LIN {X 0,Y 382.998,Z 423.777,A -85,B 0,C 180,E1 -12171.424,E2 -12171.424} C_VEL
LIN {X 0,Y 383.055,Z 423.767,A -85,B 0,C 180,E1 -12174.96,E2 -12174.96} C_VEL
LIN {X 0,Y 383.051,Z 423.767,A -85,B 0,C 180,E1 -12175.302,E2 -12175.302} C_VEL
LIN {X 0,Y 382.387,Z 423.855,A -85,B 0,C 180,E1 -12176.18,E2 -12176.18} C_VEL
LIN {X 0,Y 379.5,Z 424.21,A -85,B 0,C 180,E1 -12177.606,E2 -12177.606} C_VEL
LIN {X 0,Y 377.061,Z 424.515,A -85,B 0,C 180,E1 -12178.76,E2 -12178.76} C_VEL
LIN {X 0,Y 376.028,Z 424.643,A -85,B 0,C 180,E1 -12179.652,E2 -12179.652} C_VEL
LIN {X 0,Y 375.952,Z 424.653,A -85,B 0,C 180,E1 -12179.955,E2 -12179.955} C_VEL
LIN {X 0,Y 375.955,Z 424.652,A -85,B 0,C 180,E1 -12182.828,E2 -12182.828} C_VEL
LIN {X 0,Y 375.962,Z 424.65,A -85,B 0,C 180,E1 -12185.415,E2 -12185.415} C_VEL
LIN {X 0,Y 375.978,Z 424.653,A -85,B 0,C 180,E1 -12188.27,E2 -12188.27} C_VEL
LIN {X 0,Y 375.938,Z 424.654,A -85,B 0,C 180,E1 -12191.601,E2 -12191.601} C_VEL
LIN {X 0,Y 375.932,Z 424.654,A -85,B 0,C 180,E1 -12195.268,E2 -12195.268} C_VEL
LIN {X 0,Y 375.938,Z 424.655,A -85,B 0,C 180,E1 -12198.399,E2 -12198.399} C_VEL
LIN {X 0,Y 375.978,Z 424.652,A -85,B 0,C 180,E1 -12201.73,E2 -12201.73} C_VEL
LIN {X 0,Y 375.984,Z 424.648,A -85,B 0,C 180,E1 -12205.333,E2 -12205.333} C_VEL
LIN {X 0,Y 375.962,Z 424.651,A -85,B 0,C 180,E1 -12208.438,E2 -12208.438} C_VEL
LIN {X 0,Y 376,Z 424.649,A -85,B 0,C 180,E1 -12212.141,E2 -12212.141} C_VEL
LIN {X 0,Y 376.009,Z 424.644,A -85,B 0,C 180,E1 -12214.539,E2 -12214.539} C_VEL
LIN {X 0,Y 375.962,Z 424.654,A -85,B 0,C 180,E1 -12218.045,E2 -12218.045} C_VEL
LIN {X 0,Y 376.028,Z 424.645,A -85,B 0,C 180,E1 -12221.474,E2 -12221.474} C_VEL
LIN {X 0,Y 376.074,Z 424.74,A -85,B 0,C 180,E1 -12224.034,E2 -12224.034} C_VEL
LIN {X 0,Y 378.978,Z 436.063,A -85,B 0,C 180,E1 -12224.952,E2 -12224.952} C_VEL
LIN {X 0,Y 379.745,Z 439.16,A -85,B 0,C 180,E1 -12225.24,E2 -12225.24} C_VEL
LIN {X 0,Y 379.247,Z 450.816,A -85,B 0,C 180,E1 -12226.333,E2 -12226.333} C_VEL
LIN {X 0,Y 378.652,Z 461.215,A -85,B 0,C 180,E1 -12227.539,E2 -12227.539} C_VEL
LIN {X 0,Y 377.962,Z 471.623,A -85,B 0,C 180,E1 -12229.012,E2 -12229.012} C_VEL
LIN {X 0,Y 377.299,Z 480.79,A -85,B 0,C 180,E1 -12230.627,E2 -12230.627} C_VEL
LIN {X 0,Y 376.92,Z 488.167,A -85,B 0,C 180,E1 -12232.231,E2 -12232.231} C_VEL
LIN {X 0,Y 376.501,Z 493.226,A -85,B 0,C 180,E1 -12233.569,E2 -12233.569} C_VEL
LIN {X 0,Y 376.262,Z 498.168,A -85,B 0,C 180,E1 -12235.178,E2 -12235.178} C_VEL
LIN {X 0,Y 375.83,Z 502.008,A -85,B 0,C 180,E1 -12236.784,E2 -12236.784} C_VEL
LIN {X 0,Y 375.952,Z 503.934,A -85,B 0,C 180,E1 -12237.857,E2 -12237.857} C_VEL
LIN {X 0,Y 375.864,Z 505.478,A -85,B 0,C 180,E1 -12238.928,E2 -12238.928} C_VEL
LIN {X 0,Y 375.983,Z 506.61,A -85,B 0,C 180,E1 -12240,E2 -12240} C_VEL
LIN {X 0,Y 376.041,Z 507.304,A -85,B 0,C 180,E1 -12241.071,E2 -12241.071} C_VEL
LIN {X 0,Y 376.261,Z 507.505,A -85,B 0,C 180,E1 -12243.212,E2 -12243.212} C_VEL
LIN {X 0,Y 376.364,Z 507.004,A -85,B 0,C 180,E1 -12244.283,E2 -12244.283} C_VEL
LIN {X 0,Y 376.837,Z 504.725,A -85,B 0,C 180,E1 -12246.425,E2 -12246.425} C_VEL
LIN {X 0,Y 377.509,Z 501.851,A -85,B 0,C 180,E1 -12248.026,E2 -12248.026} C_VEL
LIN {X 0,Y 378.12,Z 497.991,A -85,B 0,C 180,E1 -12249.63,E2 -12249.63} C_VEL
LIN {X 0,Y 378.925,Z 492.952,A -85,B 0,C 180,E1 -12251.23,E2 -12251.23} C_VEL
LIN {X 0,Y 379.835,Z 486.563,A -85,B 0,C 180,E1 -12252.828,E2 -12252.828} C_VEL
LIN {X 0,Y 380.937,Z 478.602,A -85,B 0,C 180,E1 -12254.422,E2 -12254.422} C_VEL
LIN {X 0,Y 381.922,Z 470.519,A -85,B 0,C 180,E1 -12255.749,E2 -12255.749} C_VEL
LIN {X 0,Y 383.075,Z 460.593,A -85,B 0,C 180,E1 -12257.07,E2 -12257.07} C_VEL
LIN {X 0,Y 384.276,Z 449.064,A -85,B 0,C 180,E1 -12258.3,E2 -12258.3} C_VEL
LIN {X 0,Y 384.418,Z 447.136,A -85,B 0,C 180,E1 -12258.479,E2 -12258.479} C_VEL
LIN {X 0,Y 380.901,Z 436.321,A -85,B 0,C 180,E1 -12259.779,E2 -12259.779} C_VEL
LIN {X 0,Y 376.958,Z 427.479,A -85,B 0,C 180,E1 -12260.81,E2 -12260.81} C_VEL
LIN {X 0,Y 375.977,Z 424.658,A -85,B 0,C 180,E1 -12261.095,E2 -12261.095} C_VEL
LIN {X 0,Y 375.997,Z 424.649,A -85,B 0,C 180,E1 -12264.281,E2 -12264.281} C_VEL
LIN {X 0,Y 376.023,Z 424.647,A -85,B 0,C 180,E1 -12266.652,E2 -12266.652} C_VEL
LIN {X 0,Y 375.973,Z 424.653,A -85,B 0,C 180,E1 -12269.079,E2 -12269.079} C_VEL
LIN {X 0,Y 375.952,Z 424.656,A -85,B 0,C 180,E1 -12272.828,E2 -12272.828} C_VEL
LIN {X 0,Y 375.96,Z 424.653,A -85,B 0,C 180,E1 -12275.415,E2 -12275.415} C_VEL
LIN {X 0,Y 375.976,Z 424.654,A -85,B 0,C 180,E1 -12278.27,E2 -12278.27} C_VEL
LIN {X 0,Y 375.937,Z 424.652,A -85,B 0,C 180,E1 -12281.601,E2 -12281.601} C_VEL
LIN {X 0,Y 375.997,Z 424.755,A -85,B 0,C 180,E1 -12284.798,E2 -12284.798} C_VEL
LIN {X 0,Y 377.748,Z 433.032,A -85,B 0,C 180,E1 -12288.09,E2 -12288.09} C_VEL
LIN {X 0,Y 379.603,Z 442.972,A -85,B 0,C 180,E1 -12291.746,E2 -12291.746} C_VEL
LIN {X 0,Y 379.908,Z 445.692,A -85,B 0,C 180,E1 -12292.7,E2 -12292.7} C_VEL
LIN {X 0,Y 378.943,Z 454.519,A -85,B 0,C 180,E1 -12295.551,E2 -12295.551} C_VEL
LIN {X 0,Y 377.958,Z 464.839,A -85,B 0,C 180,E1 -12298.799,E2 -12298.799} C_VEL
LIN {X 0,Y 377.121,Z 475.97,A -85,B 0,C 180,E1 -12302.231,E2 -12302.231} C_VEL
LIN {X 0,Y 376.225,Z 489.228,A -85,B 0,C 180,E1 -12306.254,E2 -12306.254} C_VEL
LIN {X 0,Y 375.618,Z 500.769,A -85,B 0,C 180,E1 -12309.75,E2 -12309.75} C_VEL
LIN {X 0,Y 377.668,Z 514.335,A -85,B 0,C 180,E1 -12310.571,E2 -12310.571} C_VEL
LIN {X 0,Y 379.007,Z 537.491,A -85,B 0,C 180,E1 -12312.078,E2 -12312.078} C_VEL
LIN {X 0,Y 379.272,Z 549.569,A -85,B 0,C 180,E1 -12313.031,E2 -12313.031} C_VEL
LIN {X 0,Y 378.26,Z 560.725,A -85,B 0,C 180,E1 -12314.094,E2 -12314.094} C_VEL
LIN {X 0,Y 377.222,Z 571.102,A -85,B 0,C 180,E1 -12315.336,E2 -12315.336} C_VEL
LIN {X 0,Y 376.519,Z 579.39,A -85,B 0,C 180,E1 -12316.542,E2 -12316.542} C_VEL
LIN {X 0,Y 375.778,Z 588.341,A -85,B 0,C 180,E1 -12318.128,E2 -12318.128} C_VEL
LIN {X 0,Y 375.246,Z 595.762,A -85,B 0,C 180,E1 -12319.751,E2 -12319.751} C_VEL
LIN {X 0,Y 375.084,Z 601.755,A -85,B 0,C 180,E1 -12321.379,E2 -12321.379} C_VEL
LIN {X 0,Y 375.1,Z 607.056,A -85,B 0,C 180,E1 -12323.23,E2 -12323.23} C_VEL
LIN {X 0,Y 375.181,Z 610.145,A -85,B 0,C 180,E1 -12324.625,E2 -12324.625} C_VEL
LIN {X 0,Y 375.348,Z 611.991,A -85,B 0,C 180,E1 -12325.705,E2 -12325.705} C_VEL
LIN {X 0,Y 375.389,Z 613.39,A -85,B 0,C 180,E1 -12326.78,E2 -12326.78} C_VEL
LIN {X 0,Y 375.732,Z 614.999,A -85,B 0,C 180,E1 -12328.928,E2 -12328.928} C_VEL
LIN {X 0,Y 375.771,Z 615.131,A -85,B 0,C 180,E1 -12330,E2 -12330} C_VEL
LIN {X 0,Y 375.738,Z 614.845,A -85,B 0,C 180,E1 -12331.072,E2 -12331.072} C_VEL
LIN {X 0,Y 375.423,Z 613.021,A -85,B 0,C 180,E1 -12333.219,E2 -12333.219} C_VEL
LIN {X 0,Y 375.326,Z 610.511,A -85,B 0,C 180,E1 -12334.833,E2 -12334.833} C_VEL
LIN {X 0,Y 375.17,Z 605.883,A -85,B 0,C 180,E1 -12336.859,E2 -12336.859} C_VEL
LIN {X 0,Y 375.149,Z 600.441,A -85,B 0,C 180,E1 -12338.619,E2 -12338.619} C_VEL
LIN {X 0,Y 375.319,Z 594.079,A -85,B 0,C 180,E1 -12340.247,E2 -12340.247} C_VEL
LIN {X 0,Y 375.769,Z 586.206,A -85,B 0,C 180,E1 -12341.872,E2 -12341.872} C_VEL
LIN {X 0,Y 376.443,Z 576.913,A -85,B 0,C 180,E1 -12343.41,E2 -12343.41} C_VEL
LIN {X 0,Y 376.946,Z 570.54,A -85,B 0,C 180,E1 -12344.302,E2 -12344.302} C_VEL
LIN {X 0,Y 377.832,Z 560.218,A -85,B 0,C 180,E1 -12345.509,E2 -12345.509} C_VEL
LIN {X 0,Y 378.693,Z 550.402,A -85,B 0,C 180,E1 -12346.44,E2 -12346.44} C_VEL
LIN {X 0,Y 378.312,Z 538.497,A -85,B 0,C 180,E1 -12347.378,E2 -12347.378} C_VEL
LIN {X 0,Y 377.647,Z 525.121,A -85,B 0,C 180,E1 -12348.193,E2 -12348.193} C_VEL
LIN {X 0,Y 376.458,Z 511.651,A -85,B 0,C 180,E1 -12348.786,E2 -12348.786} C_VEL
LIN {X 0,Y 375.446,Z 503.179,A -85,B 0,C 180,E1 -12349.087,E2 -12349.087} C_VEL
LIN {X 0,Y 375.935,Z 491.639,A -85,B 0,C 180,E1 -12352.534,E2 -12352.534} C_VEL
LIN {X 0,Y 376.689,Z 478.028,A -85,B 0,C 180,E1 -12356.601,E2 -12356.601} C_VEL
LIN {X 0,Y 377.67,Z 464.562,A -85,B 0,C 180,E1 -12360.662,E2 -12360.662} C_VEL
LIN {X 0,Y 378.648,Z 452.205,A -85,B 0,C 180,E1 -12364.479,E2 -12364.479} C_VEL
LIN {X 0,Y 379.451,Z 443.597,A -85,B 0,C 180,E1 -12367.21,E2 -12367.21} C_VEL
LIN {X 0,Y 378.303,Z 436.319,A -85,B 0,C 180,E1 -12369.732,E2 -12369.732} C_VEL
LIN {X 0,Y 376.689,Z 428.211,A -85,B 0,C 180,E1 -12372.709,E2 -12372.709} C_VEL
LIN {X 0,Y 375.986,Z 424.654,A -85,B 0,C 180,E1 -12374.131,E2 -12374.131} C_VEL
LIN {X 0,Y 375.932,Z 424.66,A -85,B 0,C 180,E1 -12377.7,E2 -12377.7} C_VEL
LIN {X 0,Y 375.965,Z 424.654,A -85,B 0,C 180,E1 -12380.538,E2 -12380.538} C_VEL
LIN {X 0,Y 375.965,Z 424.651,A -85,B 0,C 180,E1 -12383.495,E2 -12383.495} C_VEL
LIN {X 0,Y 375.963,Z 424.654,A -85,B 0,C 180,E1 -12385.889,E2 -12385.889} C_VEL
LIN {X 0,Y 375.965,Z 424.652,A -85,B 0,C 180,E1 -12389.687,E2 -12389.687} C_VEL
LIN {X 0,Y 376.02,Z 424.644,A -85,B 0,C 180,E1 -12393.348,E2 -12393.348} C_VEL
LIN {X 0,Y 375.997,Z 424.647,A -85,B 0,C 180,E1 -12396.888,E2 -12396.888} C_VEL
LIN {X 0,Y 375.999,Z 424.65,A -85,B 0,C 180,E1 -12400.339,E2 -12400.339} C_VEL
LIN {X 0,Y 376.03,Z 424.645,A -85,B 0,C 180,E1 -12403.719,E2 -12403.719} C_VEL
LIN {X 0,Y 376.108,Z 424.633,A -85,B 0,C 180,E1 -12407.042,E2 -12407.042} C_VEL
LIN {X 0,Y 376.119,Z 424.635,A -85,B 0,C 180,E1 -12410.319,E2 -12410.319} C_VEL
LIN {X 0,Y 376.234,Z 424.618,A -85,B 0,C 180,E1 -12413.565,E2 -12413.565} C_VEL
LIN {X 0,Y 376.356,Z 424.606,A -85,B 0,C 180,E1 -12417.86,E2 -12417.86} C_VEL
LIN {X 0,Y 376.491,Z 424.59,A -85,B 0,C 180,E1 -12420,E2 -12420} C_VEL
LIN {X 0,Y 376.186,Z 424.623,A -85,B 0,C 180,E1 -12423.213,E2 -12423.213} C_VEL
LIN {X 0,Y 376.235,Z 424.618,A -85,B 0,C 180,E1 -12426.639,E2 -12426.639} C_VEL
LIN {X 0,Y 376.207,Z 424.621,A -85,B 0,C 180,E1 -12428.595,E2 -12428.595} C_VEL
LIN {X 0,Y 376.052,Z 424.645,A -85,B 0,C 180,E1 -12431.864,E2 -12431.864} C_VEL
LIN {X 0,Y 376.06,Z 424.639,A -85,B 0,C 180,E1 -12435.168,E2 -12435.168} C_VEL
LIN {X 0,Y 376.025,Z 424.644,A -85,B 0,C 180,E1 -12438.526,E2 -12438.526} C_VEL
LIN {X 0,Y 375.965,Z 424.656,A -85,B 0,C 180,E1 -12441.954,E2 -12441.954} C_VEL
LIN {X 0,Y 376.008,Z 424.647,A -85,B 0,C 180,E1 -12445.461,E2 -12445.461} C_VEL
LIN {X 0,Y 375.962,Z 424.651,A -85,B 0,C 180,E1 -12449.08,E2 -12449.08} C_VEL
LIN {X 0,Y 375.952,Z 424.652,A -85,B 0,C 180,E1 -12452.829,E2 -12452.829} C_VEL
LIN {X 0,Y 375.96,Z 424.653,A -85,B 0,C 180,E1 -12455.416,E2 -12455.416} C_VEL
LIN {X 0,Y 375.978,Z 424.651,A -85,B 0,C 180,E1 -12458.271,E2 -12458.271} C_VEL
LIN {X 0,Y 375.937,Z 424.658,A -85,B 0,C 180,E1 -12461.601,E2 -12461.601} C_VEL
LIN {X 0,Y 375.932,Z 424.656,A -85,B 0,C 180,E1 -12465.268,E2 -12465.268} C_VEL
LIN {X 0,Y 375.937,Z 424.655,A -85,B 0,C 180,E1 -12468.399,E2 -12468.399} C_VEL
LIN {X 0,Y 375.978,Z 424.654,A -85,B 0,C 180,E1 -12471.729,E2 -12471.729} C_VEL
LIN {X 0,Y 375.983,Z 424.65,A -85,B 0,C 180,E1 -12475.333,E2 -12475.333} C_VEL
LIN {X 0,Y 375.979,Z 424.649,A -85,B 0,C 180,E1 -12478.44,E2 -12478.44} C_VEL
LIN {X 0,Y 376.005,Z 424.648,A -85,B 0,C 180,E1 -12482.142,E2 -12482.142} C_VEL
LIN {X 0,Y 376.009,Z 424.645,A -85,B 0,C 180,E1 -12484.539,E2 -12484.539} C_VEL
LIN {X 0,Y 375.967,Z 424.653,A -85,B 0,C 180,E1 -12488.046,E2 -12488.046} C_VEL
LIN {X 0,Y 376.028,Z 424.647,A -85,B 0,C 180,E1 -12491.474,E2 -12491.474} C_VEL
LIN {X 0,Y 376.066,Z 424.642,A -85,B 0,C 180,E1 -12494.961,E2 -12494.961} C_VEL
LIN {X 0,Y 379.867,Z 437.115,A -85,B 0,C 180,E1 -12495.996,E2 -12495.996} C_VEL
LIN {X 0,Y 381.449,Z 442.817,A -85,B 0,C 180,E1 -12496.549,E2 -12496.549} C_VEL
LIN {X 0,Y 380.847,Z 453.958,A -85,B 0,C 180,E1 -12497.613,E2 -12497.613} C_VEL
LIN {X 0,Y 380.009,Z 463.886,A -85,B 0,C 180,E1 -12498.783,E2 -12498.783} C_VEL
LIN {X 0,Y 379.149,Z 473.08,A -85,B 0,C 180,E1 -12500.127,E2 -12500.127} C_VEL
LIN {X 0,Y 378.39,Z 481.826,A -85,B 0,C 180,E1 -12501.724,E2 -12501.724} C_VEL
LIN {X 0,Y 377.633,Z 488.887,A -85,B 0,C 180,E1 -12503.321,E2 -12503.321} C_VEL
LIN {X 0,Y 377.166,Z 493.645,A -85,B 0,C 180,E1 -12504.654,E2 -12504.654} C_VEL
LIN {X 0,Y 376.746,Z 498.263,A -85,B 0,C 180,E1 -12506.257,E2 -12506.257} C_VEL
LIN {X 0,Y 376.324,Z 501.822,A -85,B 0,C 180,E1 -12507.86,E2 -12507.86} C_VEL
LIN {X 0,Y 376.142,Z 503.66,A -85,B 0,C 180,E1 -12508.93,E2 -12508.93} C_VEL
LIN {X 0,Y 376.055,Z 505.047,A -85,B 0,C 180,E1 -12510,E2 -12510} C_VEL
LIN {X 0,Y 375.934,Z 506.654,A -85,B 0,C 180,E1 -12512.143,E2 -12512.143} C_VEL
LIN {X 0,Y 375.812,Z 506.92,A -85,B 0,C 180,E1 -12513.216,E2 -12513.216} C_VEL
LIN {X 0,Y 375.896,Z 506.752,A -85,B 0,C 180,E1 -12514.289,E2 -12514.289} C_VEL
LIN {X 0,Y 376.335,Z 505.236,A -85,B 0,C 180,E1 -12516.434,E2 -12516.434} C_VEL
LIN {X 0,Y 376.464,Z 503.93,A -85,B 0,C 180,E1 -12517.509,E2 -12517.509} C_VEL
LIN {X 0,Y 376.828,Z 501.14,A -85,B 0,C 180,E1 -12519.122,E2 -12519.122} C_VEL
LIN {X 0,Y 377.389,Z 497.328,A -85,B 0,C 180,E1 -12520.733,E2 -12520.733} C_VEL
LIN {X 0,Y 377.993,Z 492.406,A -85,B 0,C 180,E1 -12522.347,E2 -12522.347} C_VEL
LIN {X 0,Y 378.625,Z 486.192,A -85,B 0,C 180,E1 -12523.964,E2 -12523.964} C_VEL
LIN {X 0,Y 379.358,Z 479.664,A -85,B 0,C 180,E1 -12525.34,E2 -12525.34} C_VEL
LIN {X 0,Y 380.387,Z 470.371,A -85,B 0,C 180,E1 -12526.918,E2 -12526.918} C_VEL
LIN {X 0,Y 381.256,Z 460.584,A -85,B 0,C 180,E1 -12528.263,E2 -12528.263} C_VEL
LIN {X 0,Y 382.202,Z 449.737,A -85,B 0,C 180,E1 -12529.441,E2 -12529.441} C_VEL
LIN {X 0,Y 382.437,Z 444.949,A -85,B 0,C 180,E1 -12529.889,E2 -12529.889} C_VEL
LIN {X 0,Y 379.598,Z 435.417,A -85,B 0,C 180,E1 -12530.857,E2 -12530.857} C_VEL
LIN {X 0,Y 375.965,Z 424.653,A -85,B 0,C 180,E1 -12531.8,E2 -12531.8} C_VEL
LIN {X 0,Y 376.01,Z 424.644,A -85,B 0,C 180,E1 -12535.461,E2 -12535.461} C_VEL
LIN {X 0,Y 375.975,Z 424.648,A -85,B 0,C 180,E1 -12539.079,E2 -12539.079} C_VEL
LIN {X 0,Y 375.952,Z 424.653,A -85,B 0,C 180,E1 -12539.955,E2 -12539.955} C_VEL
LIN {X 0,Y 375.295,Z 424.74,A -85,B 0,C 180,E1 -12540.849,E2 -12540.849} C_VEL
LIN {X 0,Y 372.41,Z 425.098,A -85,B 0,C 180,E1 -12542.304,E2 -12542.304} C_VEL
LIN {X 0,Y 369.985,Z 425.395,A -85,B 0,C 180,E1 -12543.48,E2 -12543.48} C_VEL
LIN {X 0,Y 368.985,Z 425.523,A -85,B 0,C 180,E1 -12544.39,E2 -12544.39} C_VEL
LIN {X 0,Y 368.926,Z 425.526,A -85,B 0,C 180,E1 -12544.698,E2 -12544.698} C_VEL
LIN {X 0,Y 368.908,Z 425.53,A -85,B 0,C 180,E1 -12547.563,E2 -12547.563} C_VEL
LIN {X 0,Y 368.915,Z 425.532,A -85,B 0,C 180,E1 -12550.37,E2 -12550.37} C_VEL
LIN {X 0,Y 368.887,Z 425.533,A -85,B 0,C 180,E1 -12553.616,E2 -12553.616} C_VEL
LIN {X 0,Y 368.89,Z 425.532,A -85,B 0,C 180,E1 -12556.696,E2 -12556.696} C_VEL
LIN {X 0,Y 368.915,Z 425.53,A -85,B 0,C 180,E1 -12559.643,E2 -12559.643} C_VEL
LIN {X 0,Y 368.905,Z 425.529,A -85,B 0,C 180,E1 -12563.144,E2 -12563.144} C_VEL
LIN {X 0,Y 368.902,Z 425.531,A -85,B 0,C 180,E1 -12566.462,E2 -12566.462} C_VEL
LIN {X 0,Y 368.933,Z 425.526,A -85,B 0,C 180,E1 -12569.046,E2 -12569.046} C_VEL
LIN {X 0,Y 368.984,Z 425.522,A -85,B 0,C 180,E1 -12571.564,E2 -12571.564} C_VEL
LIN {X 0,Y 369.004,Z 425.521,A -85,B 0,C 180,E1 -12574.02,E2 -12574.02} C_VEL
LIN {X 0,Y 368.929,Z 425.53,A -85,B 0,C 180,E1 -12577.604,E2 -12577.604} C_VEL
LIN {X 0,Y 368.986,Z 425.52,A -85,B 0,C 180,E1 -12581.107,E2 -12581.107} C_VEL
LIN {X 0,Y 369.03,Z 425.519,A -85,B 0,C 180,E1 -12583.792,E2 -12583.792} C_VEL
LIN {X 0,Y 372.433,Z 438.96,A -85,B 0,C 180,E1 -12584.943,E2 -12584.943} C_VEL
LIN {X 0,Y 372.839,Z 441.474,A -85,B 0,C 180,E1 -12585.174,E2 -12585.174} C_VEL
LIN {X 0,Y 372.139,Z 453.389,A -85,B 0,C 180,E1 -12586.345,E2 -12586.345} C_VEL
LIN {X 0,Y 371.612,Z 463.54,A -85,B 0,C 180,E1 -12587.577,E2 -12587.577} C_VEL
LIN {X 0,Y 370.995,Z 471.979,A -85,B 0,C 180,E1 -12588.803,E2 -12588.803} C_VEL
LIN {X 0,Y 370.312,Z 481.384,A -85,B 0,C 180,E1 -12590.472,E2 -12590.472} C_VEL
LIN {X 0,Y 369.919,Z 488.736,A -85,B 0,C 180,E1 -12592.083,E2 -12592.083} C_VEL
LIN {X 0,Y 369.482,Z 493.875,A -85,B 0,C 180,E1 -12593.446,E2 -12593.446} C_VEL
LIN {X 0,Y 369.232,Z 498.907,A -85,B 0,C 180,E1 -12595.086,E2 -12595.086} C_VEL
LIN {X 0,Y 368.792,Z 502.844,A -85,B 0,C 180,E1 -12596.722,E2 -12596.722} C_VEL
LIN {X 0,Y 368.927,Z 504.844,A -85,B 0,C 180,E1 -12597.816,E2 -12597.816} C_VEL
LIN {X 0,Y 368.84,Z 506.432,A -85,B 0,C 180,E1 -12598.908,E2 -12598.908} C_VEL
LIN {X 0,Y 368.966,Z 507.61,A -85,B 0,C 180,E1 -12600,E2 -12600} C_VEL
LIN {X 0,Y 369.028,Z 508.374,A -85,B 0,C 180,E1 -12601.091,E2 -12601.091} C_VEL
LIN {X 0,Y 369.152,Z 508.703,A -85,B 0,C 180,E1 -12602.182,E2 -12602.182} C_VEL
LIN {X 0,Y 369.275,Z 508.653,A -85,B 0,C 180,E1 -12603.273,E2 -12603.273} C_VEL
LIN {X 0,Y 369.385,Z 508.216,A -85,B 0,C 180,E1 -12604.365,E2 -12604.365} C_VEL
LIN {X 0,Y 369.905,Z 506.039,A -85,B 0,C 180,E1 -12606.546,E2 -12606.546} C_VEL
LIN {X 0,Y 370.63,Z 503.262,A -85,B 0,C 180,E1 -12608.176,E2 -12608.176} C_VEL
LIN {X 0,Y 371.28,Z 499.481,A -85,B 0,C 180,E1 -12609.809,E2 -12609.809} C_VEL
LIN {X 0,Y 372.146,Z 494.534,A -85,B 0,C 180,E1 -12611.437,E2 -12611.437} C_VEL
LIN {X 0,Y 373.133,Z 488.278,A -85,B 0,C 180,E1 -12613.063,E2 -12613.063} C_VEL
LIN {X 0,Y 374.328,Z 480.505,A -85,B 0,C 180,E1 -12614.682,E2 -12614.682} C_VEL
LIN {X 0,Y 375.379,Z 472.598,A -85,B 0,C 180,E1 -12616.031,E2 -12616.031} C_VEL
LIN {X 0,Y 376.589,Z 462.892,A -85,B 0,C 180,E1 -12617.373,E2 -12617.373} C_VEL
LIN {X 0,Y 377.874,Z 451.542,A -85,B 0,C 180,E1 -12618.641,E2 -12618.641} C_VEL
LIN {X 0,Y 378.064,Z 449.476,A -85,B 0,C 180,E1 -12618.84,E2 -12618.84} C_VEL
LIN {X 0,Y 375.264,Z 440.491,A -85,B 0,C 180,E1 -12619.986,E2 -12619.986} C_VEL
LIN {X 0,Y 370.695,Z 429.697,A -85,B 0,C 180,E1 -12621.328,E2 -12621.328} C_VEL
LIN {X 0,Y 369.043,Z 426.27,A -85,B 0,C 180,E1 -12621.741,E2 -12621.741} C_VEL
LIN {X 0,Y 368.941,Z 425.536,A -85,B 0,C 180,E1 -12621.805,E2 -12621.805} C_VEL
LIN {X 0,Y 368.961,Z 425.527,A -85,B 0,C 180,E1 -12624.775,E2 -12624.775} C_VEL
LIN {X 0,Y 368.971,Z 425.526,A -85,B 0,C 180,E1 -12627.203,E2 -12627.203} C_VEL
LIN {X 0,Y 368.922,Z 425.529,A -85,B 0,C 180,E1 -12629.69,E2 -12629.69} C_VEL
LIN {X 0,Y 368.9,Z 425.533,A -85,B 0,C 180,E1 -12633.043,E2 -12633.043} C_VEL
LIN {X 0,Y 368.92,Z 425.532,A -85,B 0,C 180,E1 -12636.197,E2 -12636.197} C_VEL
LIN {X 0,Y 368.905,Z 425.532,A -85,B 0,C 180,E1 -12638.953,E2 -12638.953} C_VEL
LIN {X 0,Y 368.883,Z 425.531,A -85,B 0,C 180,E1 -12642.009,E2 -12642.009} C_VEL
LIN {X 0,Y 368.924,Z 425.588,A -85,B 0,C 180,E1 -12644.328,E2 -12644.328} C_VEL
LIN {X 0,Y 370.894,Z 434.784,A -85,B 0,C 180,E1 -12648.077,E2 -12648.077} C_VEL
LIN {X 0,Y 372.544,Z 443.871,A -85,B 0,C 180,E1 -12651.498,E2 -12651.498} C_VEL
LIN {X 0,Y 372.941,Z 446.174,A -85,B 0,C 180,E1 -12652.324,E2 -12652.324} C_VEL
LIN {X 0,Y 372.168,Z 453.768,A -85,B 0,C 180,E1 -12654.853,E2 -12654.853} C_VEL
LIN {X 0,Y 371.047,Z 464.964,A -85,B 0,C 180,E1 -12658.468,E2 -12658.468} C_VEL
LIN {X 0,Y 370.034,Z 477.018,A -85,B 0,C 180,E1 -12662.268,E2 -12662.268} C_VEL
LIN {X 0,Y 369.173,Z 489.138,A -85,B 0,C 180,E1 -12666.034,E2 -12666.034} C_VEL
LIN {X 0,Y 368.627,Z 499.227,A -85,B 0,C 180,E1 -12669.1,E2 -12669.1} C_VEL
LIN {X 0,Y 370.992,Z 513.976,A -85,B 0,C 180,E1 -12670.063,E2 -12670.063} C_VEL
LIN {X 0,Y 371.818,Z 528.383,A -85,B 0,C 180,E1 -12671.106,E2 -12671.106} C_VEL
LIN {X 0,Y 372.226,Z 545.56,A -85,B 0,C 180,E1 -12672.416,E2 -12672.416} C_VEL
LIN {X 0,Y 372.14,Z 553.252,A -85,B 0,C 180,E1 -12673.12,E2 -12673.12} C_VEL
LIN {X 0,Y 370.857,Z 564.617,A -85,B 0,C 180,E1 -12674.333,E2 -12674.333} C_VEL
LIN {X 0,Y 369.827,Z 575.003,A -85,B 0,C 180,E1 -12675.738,E2 -12675.738} C_VEL
LIN {X 0,Y 369.136,Z 583.091,A -85,B 0,C 180,E1 -12677.073,E2 -12677.073} C_VEL
LIN {X 0,Y 368.46,Z 591.318,A -85,B 0,C 180,E1 -12678.725,E2 -12678.725} C_VEL
LIN {X 0,Y 368.123,Z 596.936,A -85,B 0,C 180,E1 -12680.106,E2 -12680.106} C_VEL
LIN {X 0,Y 368.006,Z 602.482,A -85,B 0,C 180,E1 -12681.765,E2 -12681.765} C_VEL
LIN {X 0,Y 368.058,Z 606.842,A -85,B 0,C 180,E1 -12683.421,E2 -12683.421} C_VEL
LIN {X 0,Y 368.111,Z 609.161,A -85,B 0,C 180,E1 -12684.522,E2 -12684.522} C_VEL
LIN {X 0,Y 368.277,Z 610.998,A -85,B 0,C 180,E1 -12685.622,E2 -12685.622} C_VEL
LIN {X 0,Y 368.339,Z 612.395,A -85,B 0,C 180,E1 -12686.718,E2 -12686.718} C_VEL
LIN {X 0,Y 368.702,Z 613.992,A -85,B 0,C 180,E1 -12688.908,E2 -12688.908} C_VEL
LIN {X 0,Y 368.748,Z 614.116,A -85,B 0,C 180,E1 -12690,E2 -12690} C_VEL
LIN {X 0,Y 368.709,Z 613.822,A -85,B 0,C 180,E1 -12691.092,E2 -12691.092} C_VEL
LIN {X 0,Y 368.38,Z 611.98,A -85,B 0,C 180,E1 -12693.281,E2 -12693.281} C_VEL
LIN {X 0,Y 368.266,Z 609.455,A -85,B 0,C 180,E1 -12694.926,E2 -12694.926} C_VEL
LIN {X 0,Y 368.097,Z 605.135,A -85,B 0,C 180,E1 -12696.866,E2 -12696.866} C_VEL
LIN {X 0,Y 368.072,Z 599.336,A -85,B 0,C 180,E1 -12698.786,E2 -12698.786} C_VEL
LIN {X 0,Y 368.258,Z 592.954,A -85,B 0,C 180,E1 -12700.445,E2 -12700.445} C_VEL
LIN {X 0,Y 368.76,Z 585.055,A -85,B 0,C 180,E1 -12702.101,E2 -12702.101} C_VEL
LIN {X 0,Y 369.373,Z 576.241,A -85,B 0,C 180,E1 -12703.592,E2 -12703.592} C_VEL
LIN {X 0,Y 370.252,Z 567.196,A -85,B 0,C 180,E1 -12704.848,E2 -12704.848} C_VEL
LIN {X 0,Y 371.163,Z 556.345,A -85,B 0,C 180,E1 -12706.077,E2 -12706.077} C_VEL
LIN {X 0,Y 371.695,Z 549.079,A -85,B 0,C 180,E1 -12706.759,E2 -12706.759} C_VEL
LIN {X 0,Y 371.319,Z 537.235,A -85,B 0,C 180,E1 -12707.707,E2 -12707.707} C_VEL
LIN {X 0,Y 370.607,Z 524.052,A -85,B 0,C 180,E1 -12708.527,E2 -12708.527} C_VEL
LIN {X 0,Y 369.414,Z 510.776,A -85,B 0,C 180,E1 -12709.126,E2 -12709.126} C_VEL
LIN {X 0,Y 368.408,Z 502.192,A -85,B 0,C 180,E1 -12709.429,E2 -12709.429} C_VEL
LIN {X 0,Y 368.901,Z 490.544,A -85,B 0,C 180,E1 -12712.989,E2 -12712.989} C_VEL
LIN {X 0,Y 369.64,Z 478.527,A -85,B 0,C 180,E1 -12716.669,E2 -12716.669} C_VEL
LIN {X 0,Y 370.643,Z 465.167,A -85,B 0,C 180,E1 -12720.795,E2 -12720.795} C_VEL
LIN {X 0,Y 371.651,Z 453.24,A -85,B 0,C 180,E1 -12724.562,E2 -12724.562} C_VEL
LIN {X 0,Y 372.461,Z 445.265,A -85,B 0,C 180,E1 -12727.143,E2 -12727.143} C_VEL
LIN {X 0,Y 371.689,Z 439.455,A -85,B 0,C 180,E1 -12729.173,E2 -12729.173} C_VEL
LIN {X 0,Y 370.092,Z 431.225,A -85,B 0,C 180,E1 -12732.217,E2 -12732.217} C_VEL
LIN {X 0,Y 368.917,Z 425.537,A -85,B 0,C 180,E1 -12734.501,E2 -12734.501} C_VEL
LIN {X 0,Y 368.884,Z 425.538,A -85,B 0,C 180,E1 -12738.178,E2 -12738.178} C_VEL
LIN {X 0,Y 368.911,Z 425.529,A -85,B 0,C 180,E1 -12741.359,E2 -12741.359} C_VEL
LIN {X 0,Y 368.937,Z 425.525,A -85,B 0,C 180,E1 -12745.147,E2 -12745.147} C_VEL
LIN {X 0,Y 368.929,Z 425.527,A -85,B 0,C 180,E1 -12749.047,E2 -12749.047} C_VEL
LIN {X 0,Y 368.964,Z 425.523,A -85,B 0,C 180,E1 -12752.797,E2 -12752.797} C_VEL
LIN {X 0,Y 368.946,Z 425.53,A -85,B 0,C 180,E1 -12756.113,E2 -12756.113} C_VEL
LIN {X 0,Y 368.938,Z 425.53,A -85,B 0,C 180,E1 -12759.947,E2 -12759.947} C_VEL
LIN {X 0,Y 368.977,Z 425.521,A -85,B 0,C 180,E1 -12763.399,E2 -12763.399} C_VEL
LIN {X 0,Y 369.061,Z 425.511,A -85,B 0,C 180,E1 -12766.79,E2 -12766.79} C_VEL
LIN {X 0,Y 369.069,Z 425.515,A -85,B 0,C 180,E1 -12770.132,E2 -12770.132} C_VEL
LIN {X 0,Y 369.192,Z 425.494,A -85,B 0,C 180,E1 -12773.442,E2 -12773.442} C_VEL
LIN {X 0,Y 369.321,Z 425.482,A -85,B 0,C 180,E1 -12777.819,E2 -12777.819} C_VEL
LIN {X 0,Y 369.46,Z 425.466,A -85,B 0,C 180,E1 -12780,E2 -12780} C_VEL
LIN {X 0,Y 369.318,Z 425.483,A -85,B 0,C 180,E1 -12782.181,E2 -12782.181} C_VEL
LIN {X 0,Y 369.205,Z 425.493,A -85,B 0,C 180,E1 -12786.627,E2 -12786.627} C_VEL
LIN {X 0,Y 369.139,Z 425.501,A -85,B 0,C 180,E1 -12788.761,E2 -12788.761} C_VEL
LIN {X 0,Y 369.008,Z 425.522,A -85,B 0,C 180,E1 -12792.093,E2 -12792.093} C_VEL
LIN {X 0,Y 368.999,Z 425.519,A -85,B 0,C 180,E1 -12795.465,E2 -12795.465} C_VEL
LIN {X 0,Y 368.984,Z 425.52,A -85,B 0,C 180,E1 -12798.893,E2 -12798.893} C_VEL
LIN {X 0,Y 368.934,Z 425.528,A -85,B 0,C 180,E1 -12802.395,E2 -12802.395} C_VEL
LIN {X 0,Y 369.001,Z 425.523,A -85,B 0,C 180,E1 -12805.98,E2 -12805.98} C_VEL
LIN {X 0,Y 368.916,Z 425.532,A -85,B 0,C 180,E1 -12809.691,E2 -12809.691} C_VEL
LIN {X 0,Y 368.9,Z 425.53,A -85,B 0,C 180,E1 -12813.044,E2 -12813.044} C_VEL
LIN {X 0,Y 368.92,Z 425.531,A -85,B 0,C 180,E1 -12816.197,E2 -12816.197} C_VEL
LIN {X 0,Y 368.906,Z 425.529,A -85,B 0,C 180,E1 -12818.953,E2 -12818.953} C_VEL
LIN {X 0,Y 368.884,Z 425.537,A -85,B 0,C 180,E1 -12822.01,E2 -12822.01} C_VEL
LIN {X 0,Y 368.885,Z 425.533,A -85,B 0,C 180,E1 -12825.177,E2 -12825.177} C_VEL
LIN {X 0,Y 368.886,Z 425.535,A -85,B 0,C 180,E1 -12828.178,E2 -12828.178} C_VEL
LIN {X 0,Y 368.912,Z 425.531,A -85,B 0,C 180,E1 -12831.36,E2 -12831.36} C_VEL
LIN {X 0,Y 368.939,Z 425.526,A -85,B 0,C 180,E1 -12835.147,E2 -12835.147} C_VEL
LIN {X 0,Y 368.932,Z 425.527,A -85,B 0,C 180,E1 -12839.047,E2 -12839.047} C_VEL
LIN {X 0,Y 368.99,Z 425.524,A -85,B 0,C 180,E1 -12841.565,E2 -12841.565} C_VEL
LIN {X 0,Y 368.961,Z 425.524,A -85,B 0,C 180,E1 -12845.225,E2 -12845.225} C_VEL
LIN {X 0,Y 368.941,Z 425.526,A -85,B 0,C 180,E1 -12848.974,E2 -12848.974} C_VEL
LIN {X 0,Y 368.994,Z 425.52,A -85,B 0,C 180,E1 -12852.258,E2 -12852.258} C_VEL
LIN {X 0,Y 369.027,Z 425.634,A -85,B 0,C 180,E1 -12854.635,E2 -12854.635} C_VEL
LIN {X 0,Y 372.753,Z 437.637,A -85,B 0,C 180,E1 -12855.642,E2 -12855.642} C_VEL
LIN {X 0,Y 374.612,Z 444.234,A -85,B 0,C 180,E1 -12856.299,E2 -12856.299} C_VEL
LIN {X 0,Y 374.014,Z 455.295,A -85,B 0,C 180,E1 -12857.383,E2 -12857.383} C_VEL
LIN {X 0,Y 373.149,Z 465.158,A -85,B 0,C 180,E1 -12858.574,E2 -12858.574} C_VEL
LIN {X 0,Y 372.253,Z 474.295,A -85,B 0,C 180,E1 -12859.943,E2 -12859.943} C_VEL
LIN {X 0,Y 371.461,Z 483.007,A -85,B 0,C 180,E1 -12861.569,E2 -12861.569} C_VEL
LIN {X 0,Y 370.672,Z 490.038,A -85,B 0,C 180,E1 -12863.195,E2 -12863.195} C_VEL
LIN {X 0,Y 370.213,Z 494.765,A -85,B 0,C 180,E1 -12864.554,E2 -12864.554} C_VEL
LIN {X 0,Y 369.753,Z 499.363,A -85,B 0,C 180,E1 -12866.186,E2 -12866.186} C_VEL
LIN {X 0,Y 369.308,Z 502.901,A -85,B 0,C 180,E1 -12867.819,E2 -12867.819} C_VEL
LIN {X 0,Y 369.121,Z 504.726,A -85,B 0,C 180,E1 -12868.909,E2 -12868.909} C_VEL
LIN {X 0,Y 368.981,Z 507.069,A -85,B 0,C 180,E1 -12871.092,E2 -12871.092} C_VEL
LIN {X 0,Y 368.91,Z 507.681,A -85,B 0,C 180,E1 -12872.184,E2 -12872.184} C_VEL
LIN {X 0,Y 368.788,Z 507.936,A -85,B 0,C 180,E1 -12873.278,E2 -12873.278} C_VEL
LIN {X 0,Y 369.046,Z 507.174,A -85,B 0,C 180,E1 -12875.464,E2 -12875.464} C_VEL
LIN {X 0,Y 369.346,Z 506.212,A -85,B 0,C 180,E1 -12876.556,E2 -12876.556} C_VEL
LIN {X 0,Y 369.488,Z 504.894,A -85,B 0,C 180,E1 -12877.652,E2 -12877.652} C_VEL
LIN {X 0,Y 369.885,Z 502.085,A -85,B 0,C 180,E1 -12879.294,E2 -12879.294} C_VEL
LIN {X 0,Y 370.461,Z 498.252,A -85,B 0,C 180,E1 -12880.936,E2 -12880.936} C_VEL
LIN {X 0,Y 371.11,Z 493.303,A -85,B 0,C 180,E1 -12882.579,E2 -12882.579} C_VEL
LIN {X 0,Y 371.786,Z 487.049,A -85,B 0,C 180,E1 -12884.226,E2 -12884.226} C_VEL
LIN {X 0,Y 372.777,Z 478.774,A -85,B 0,C 180,E1 -12885.947,E2 -12885.947} C_VEL
LIN {X 0,Y 373.83,Z 469.381,A -85,B 0,C 180,E1 -12887.506,E2 -12887.506} C_VEL
LIN {X 0,Y 374.67,Z 460.177,A -85,B 0,C 180,E1 -12888.738,E2 -12888.738} C_VEL
LIN {X 0,Y 375.601,Z 449.67,A -85,B 0,C 180,E1 -12889.869,E2 -12889.869} C_VEL
LIN {X 0,Y 375.713,Z 446.52,A -85,B 0,C 180,E1 -12890.174,E2 -12890.174} C_VEL
LIN {X 0,Y 372.201,Z 435.095,A -85,B 0,C 180,E1 -12891.357,E2 -12891.357} C_VEL
LIN {X 0,Y 368.924,Z 425.532,A -85,B 0,C 180,E1 -12892.215,E2 -12892.215} C_VEL
LIN {X 0,Y 369.004,Z 425.52,A -85,B 0,C 180,E1 -12895.98,E2 -12895.98} C_VEL
LIN {X 0,Y 368.965,Z 425.523,A -85,B 0,C 180,E1 -12898.812,E2 -12898.812} C_VEL
LIN {X 0,Y 368.903,Z 425.536,A -85,B 0,C 180,E1 -12902.238,E2 -12902.238} C_VEL
LIN {X 0,Y 368.926,Z 425.526,A -85,B 0,C 180,E1 -12904.698,E2 -12904.698} C_VEL
LIN {X 0,Y 368.314,Z 425.606,A -85,B 0,C 180,E1 -12905.609,E2 -12905.609} C_VEL
LIN {X 0,Y 365.457,Z 425.961,A -85,B 0,C 180,E1 -12907.089,E2 -12907.089} C_VEL
LIN {X 0,Y 362.999,Z 426.27,A -85,B 0,C 180,E1 -12908.286,E2 -12908.286} C_VEL
LIN {X 0,Y 361.941,Z 426.397,A -85,B 0,C 180,E1 -12909.213,E2 -12909.213} C_VEL
LIN {X 0,Y 361.855,Z 426.408,A -85,B 0,C 180,E1 -12909.527,E2 -12909.527} C_VEL
LIN {X 0,Y 361.84,Z 426.409,A -85,B 0,C 180,E1 -12912.829,E2 -12912.829} C_VEL
LIN {X 0,Y 361.823,Z 426.416,A -85,B 0,C 180,E1 -12915.946,E2 -12915.946} C_VEL
LIN {X 0,Y 361.839,Z 426.409,A -85,B 0,C 180,E1 -12919.245,E2 -12919.245} C_VEL
LIN {X 0,Y 361.868,Z 426.406,A -85,B 0,C 180,E1 -12922.777,E2 -12922.777} C_VEL
LIN {X 0,Y 361.859,Z 426.411,A -85,B 0,C 180,E1 -12925.72,E2 -12925.72} C_VEL
LIN {X 0,Y 361.879,Z 426.408,A -85,B 0,C 180,E1 -12929.672,E2 -12929.672} C_VEL
LIN {X 0,Y 361.958,Z 426.397,A -85,B 0,C 180,E1 -12933.475,E2 -12933.475} C_VEL
LIN {X 0,Y 361.886,Z 426.404,A -85,B 0,C 180,E1 -12937.144,E2 -12937.144} C_VEL
LIN {X 0,Y 361.925,Z 426.398,A -85,B 0,C 180,E1 -12940.724,E2 -12940.724} C_VEL
LIN {X 0,Y 361.995,Z 426.431,A -85,B 0,C 180,E1 -12943.613,E2 -12943.613} C_VEL
LIN {X 0,Y 365.046,Z 438.518,A -85,B 0,C 180,E1 -12944.631,E2 -12944.631} C_VEL
LIN {X 0,Y 365.865,Z 442.716,A -85,B 0,C 180,E1 -12945.029,E2 -12945.029} C_VEL
LIN {X 0,Y 365.138,Z 454.527,A -85,B 0,C 180,E1 -12946.22,E2 -12946.22} C_VEL
LIN {X 0,Y 364.597,Z 464.649,A -85,B 0,C 180,E1 -12947.475,E2 -12947.475} C_VEL
LIN {X 0,Y 363.895,Z 473.92,A -85,B 0,C 180,E1 -12948.864,E2 -12948.864} C_VEL
LIN {X 0,Y 363.316,Z 481.97,A -85,B 0,C 180,E1 -12950.324,E2 -12950.324} C_VEL
LIN {X 0,Y 362.919,Z 489.262,A -85,B 0,C 180,E1 -12951.929,E2 -12951.929} C_VEL
LIN {X 0,Y 362.466,Z 494.509,A -85,B 0,C 180,E1 -12953.319,E2 -12953.319} C_VEL
LIN {X 0,Y 362.208,Z 499.641,A -85,B 0,C 180,E1 -12954.991,E2 -12954.991} C_VEL
LIN {X 0,Y 361.753,Z 503.673,A -85,B 0,C 180,E1 -12956.659,E2 -12956.659} C_VEL
LIN {X 0,Y 361.9,Z 505.752,A -85,B 0,C 180,E1 -12957.774,E2 -12957.774} C_VEL
LIN {X 0,Y 361.815,Z 507.389,A -85,B 0,C 180,E1 -12958.887,E2 -12958.887} C_VEL
LIN {X 0,Y 361.948,Z 508.605,A -85,B 0,C 180,E1 -12960,E2 -12960} C_VEL
LIN {X 0,Y 362.014,Z 509.44,A -85,B 0,C 180,E1 -12961.112,E2 -12961.112} C_VEL
LIN {X 0,Y 362.146,Z 509.822,A -85,B 0,C 180,E1 -12962.224,E2 -12962.224} C_VEL
LIN {X 0,Y 362.434,Z 509.442,A -85,B 0,C 180,E1 -12964.448,E2 -12964.448} C_VEL
LIN {X 0,Y 362.674,Z 508.617,A -85,B 0,C 180,E1 -12965.56,E2 -12965.56} C_VEL
LIN {X 0,Y 362.992,Z 507.372,A -85,B 0,C 180,E1 -12966.671,E2 -12966.671} C_VEL
LIN {X 0,Y 363.748,Z 504.674,A -85,B 0,C 180,E1 -12968.332,E2 -12968.332} C_VEL
LIN {X 0,Y 364.446,Z 500.985,A -85,B 0,C 180,E1 -12969.995,E2 -12969.995} C_VEL
LIN {X 0,Y 365.393,Z 496.173,A -85,B 0,C 180,E1 -12971.651,E2 -12971.651} C_VEL
LIN {X 0,Y 366.467,Z 490.095,A -85,B 0,C 180,E1 -12973.305,E2 -12973.305} C_VEL
LIN {X 0,Y 367.728,Z 482.439,A -85,B 0,C 180,E1 -12974.952,E2 -12974.952} C_VEL
LIN {X 0,Y 369.078,Z 472.99,A -85,B 0,C 180,E1 -12976.596,E2 -12976.596} C_VEL
LIN {X 0,Y 370.322,Z 463.898,A -85,B 0,C 180,E1 -12977.87,E2 -12977.87} C_VEL
LIN {X 0,Y 371.745,Z 452.318,A -85,B 0,C 180,E1 -12979.179,E2 -12979.179} C_VEL
LIN {X 0,Y 369.318,Z 443.699,A -85,B 0,C 180,E1 -12980.322,E2 -12980.322} C_VEL
LIN {X 0,Y 365.526,Z 434.468,A -85,B 0,C 180,E1 -12981.55,E2 -12981.55} C_VEL
LIN {X 0,Y 362.211,Z 427.729,A -85,B 0,C 180,E1 -12982.449,E2 -12982.449} C_VEL
LIN {X 0,Y 361.9,Z 426.408,A -85,B 0,C 180,E1 -12982.591,E2 -12982.591} C_VEL
LIN {X 0,Y 361.958,Z 426.398,A -85,B 0,C 180,E1 -12986.525,E2 -12986.525} C_VEL
LIN {X 0,Y 361.877,Z 426.409,A -85,B 0,C 180,E1 -12990.328,E2 -12990.328} C_VEL
LIN {X 0,Y 361.857,Z 426.412,A -85,B 0,C 180,E1 -12994.28,E2 -12994.28} C_VEL
LIN {X 0,Y 361.866,Z 426.408,A -85,B 0,C 180,E1 -12997.223,E2 -12997.223} C_VEL
LIN {X 0,Y 361.838,Z 426.413,A -85,B 0,C 180,E1 -13000.755,E2 -13000.755} C_VEL
LIN {X 0,Y 361.86,Z 426.437,A -85,B 0,C 180,E1 -13003.868,E2 -13003.868} C_VEL
LIN {X 0,Y 363.672,Z 434.964,A -85,B 0,C 180,E1 -13007.438,E2 -13007.438} C_VEL
LIN {X 0,Y 365.396,Z 444.028,A -85,B 0,C 180,E1 -13010.956,E2 -13010.956} C_VEL
LIN {X 0,Y 365.907,Z 447.054,A -85,B 0,C 180,E1 -13012.075,E2 -13012.075} C_VEL
LIN {X 0,Y 365.706,Z 450.95,A -85,B 0,C 180,E1 -13013.434,E2 -13013.434} C_VEL
LIN {X 0,Y 364.396,Z 462.6,A -85,B 0,C 180,E1 -13017.314,E2 -13017.314} C_VEL
LIN {X 0,Y 363.27,Z 474.195,A -85,B 0,C 180,E1 -13021.075,E2 -13021.075} C_VEL
LIN {X 0,Y 362.371,Z 485.688,A -85,B 0,C 180,E1 -13024.743,E2 -13024.743} C_VEL
LIN {X 0,Y 361.644,Z 497.073,A -85,B 0,C 180,E1 -13028.356,E2 -13028.356} C_VEL
LIN {X 0,Y 364.177,Z 512.043,A -85,B 0,C 180,E1 -13029.407,E2 -13029.407} C_VEL
LIN {X 0,Y 364.98,Z 522.786,A -85,B 0,C 180,E1 -13030.204,E2 -13030.204} C_VEL
LIN {X 0,Y 365.245,Z 536.879,A -85,B 0,C 180,E1 -13031.401,E2 -13031.401} C_VEL
LIN {X 0,Y 365.37,Z 551.016,A -85,B 0,C 180,E1 -13032.653,E2 -13032.653} C_VEL
LIN {X 0,Y 364.153,Z 562.636,A -85,B 0,C 180,E1 -13033.893,E2 -13033.893} C_VEL
LIN {X 0,Y 363.137,Z 572.037,A -85,B 0,C 180,E1 -13035.141,E2 -13035.141} C_VEL
LIN {X 0,Y 362.404,Z 579.584,A -85,B 0,C 180,E1 -13036.349,E2 -13036.349} C_VEL
LIN {X 0,Y 361.649,Z 587.856,A -85,B 0,C 180,E1 -13037.941,E2 -13037.941} C_VEL
LIN {X 0,Y 361.096,Z 594.94,A -85,B 0,C 180,E1 -13039.628,E2 -13039.628} C_VEL
LIN {X 0,Y 360.926,Z 601.518,A -85,B 0,C 180,E1 -13041.602,E2 -13041.602} C_VEL
LIN {X 0,Y 360.969,Z 605.865,A -85,B 0,C 180,E1 -13043.291,E2 -13043.291} C_VEL
LIN {X 0,Y 361.043,Z 608.178,A -85,B 0,C 180,E1 -13044.414,E2 -13044.414} C_VEL
LIN {X 0,Y 361.209,Z 610.006,A -85,B 0,C 180,E1 -13045.536,E2 -13045.536} C_VEL
LIN {X 0,Y 361.289,Z 611.4,A -85,B 0,C 180,E1 -13046.654,E2 -13046.654} C_VEL
LIN {X 0,Y 361.671,Z 612.984,A -85,B 0,C 180,E1 -13048.886,E2 -13048.886} C_VEL
LIN {X 0,Y 361.724,Z 613.101,A -85,B 0,C 180,E1 -13050,E2 -13050} C_VEL
LIN {X 0,Y 361.679,Z 612.8,A -85,B 0,C 180,E1 -13051.113,E2 -13051.113} C_VEL
LIN {X 0,Y 361.335,Z 610.937,A -85,B 0,C 180,E1 -13053.345,E2 -13053.345} C_VEL
LIN {X 0,Y 361.205,Z 608.397,A -85,B 0,C 180,E1 -13055.023,E2 -13055.023} C_VEL
LIN {X 0,Y 361.036,Z 604.346,A -85,B 0,C 180,E1 -13056.89,E2 -13056.89} C_VEL
LIN {X 0,Y 361.016,Z 598.233,A -85,B 0,C 180,E1 -13058.959,E2 -13058.959} C_VEL
LIN {X 0,Y 361.218,Z 591.83,A -85,B 0,C 180,E1 -13060.651,E2 -13060.651} C_VEL
LIN {X 0,Y 361.713,Z 583.893,A -85,B 0,C 180,E1 -13062.341,E2 -13062.341} C_VEL
LIN {X 0,Y 362.306,Z 576.088,A -85,B 0,C 180,E1 -13063.701,E2 -13063.701} C_VEL
LIN {X 0,Y 363.235,Z 567.075,A -85,B 0,C 180,E1 -13064.998,E2 -13064.998} C_VEL
LIN {X 0,Y 364.165,Z 556.407,A -85,B 0,C 180,E1 -13066.25,E2 -13066.25} C_VEL
LIN {X 0,Y 364.672,Z 549.359,A -85,B 0,C 180,E1 -13066.947,E2 -13066.947} C_VEL
LIN {X 0,Y 364.33,Z 536.96,A -85,B 0,C 180,E1 -13067.977,E2 -13067.977} C_VEL
LIN {X 0,Y 363.678,Z 523.865,A -85,B 0,C 180,E1 -13068.82,E2 -13068.82} C_VEL
LIN {X 0,Y 362.547,Z 510.946,A -85,B 0,C 180,E1 -13069.439,E2 -13069.439} C_VEL
LIN {X 0,Y 361.352,Z 501.2,A -85,B 0,C 180,E1 -13069.788,E2 -13069.788} C_VEL
LIN {X 0,Y 361.891,Z 489.463,A -85,B 0,C 180,E1 -13073.46,E2 -13073.46} C_VEL
LIN {X 0,Y 362.674,Z 477.345,A -85,B 0,C 180,E1 -13077.265,E2 -13077.265} C_VEL
LIN {X 0,Y 363.767,Z 464.151,A -85,B 0,C 180,E1 -13081.442,E2 -13081.442} C_VEL
LIN {X 0,Y 364.908,Z 452.266,A -85,B 0,C 180,E1 -13085.295,E2 -13085.295} C_VEL
LIN {X 0,Y 365.498,Z 446.375,A -85,B 0,C 180,E1 -13087.252,E2 -13087.252} C_VEL
LIN {X 0,Y 364.792,Z 441.131,A -85,B 0,C 180,E1 -13089.12,E2 -13089.12} C_VEL
LIN {X 0,Y 363.366,Z 433.813,A -85,B 0,C 180,E1 -13091.871,E2 -13091.871} C_VEL
LIN {X 0,Y 361.888,Z 426.413,A -85,B 0,C 180,E1 -13094.876,E2 -13094.876} C_VEL
LIN {X 0,Y 361.828,Z 426.413,A -85,B 0,C 180,E1 -13098.669,E2 -13098.669} C_VEL
LIN {X 0,Y 361.873,Z 426.406,A -85,B 0,C 180,E1 -13101.576,E2 -13101.576} C_VEL
LIN {X 0,Y 361.875,Z 426.407,A -85,B 0,C 180,E1 -13104.655,E2 -13104.655} C_VEL
LIN {X 0,Y 361.838,Z 426.414,A -85,B 0,C 180,E1 -13108.371,E2 -13108.371} C_VEL
LIN {X 0,Y 361.909,Z 426.407,A -85,B 0,C 180,E1 -13112.221,E2 -13112.221} C_VEL
LIN {X 0,Y 361.929,Z 426.4,A -85,B 0,C 180,E1 -13114.71,E2 -13114.71} C_VEL
LIN {X 0,Y 361.892,Z 426.407,A -85,B 0,C 180,E1 -13118.347,E2 -13118.347} C_VEL
LIN {X 0,Y 361.968,Z 426.399,A -85,B 0,C 180,E1 -13122.061,E2 -13122.061} C_VEL
LIN {X 0,Y 361.999,Z 426.396,A -85,B 0,C 180,E1 -13126.101,E2 -13126.101} C_VEL
LIN {X 0,Y 362.034,Z 426.39,A -85,B 0,C 180,E1 -13129.938,E2 -13129.938} C_VEL
LIN {X 0,Y 362.153,Z 426.371,A -85,B 0,C 180,E1 -13133.314,E2 -13133.314} C_VEL
LIN {X 0,Y 362.285,Z 426.357,A -85,B 0,C 180,E1 -13137.777,E2 -13137.777} C_VEL
LIN {X 0,Y 362.429,Z 426.342,A -85,B 0,C 180,E1 -13140,E2 -13140} C_VEL
LIN {X 0,Y 362.282,Z 426.359,A -85,B 0,C 180,E1 -13142.224,E2 -13142.224} C_VEL
LIN {X 0,Y 362.174,Z 426.368,A -85,B 0,C 180,E1 -13146.686,E2 -13146.686} C_VEL
LIN {X 0,Y 362.075,Z 426.38,A -85,B 0,C 180,E1 -13148.933,E2 -13148.933} C_VEL
LIN {X 0,Y 361.962,Z 426.397,A -85,B 0,C 180,E1 -13152.332,E2 -13152.332} C_VEL
LIN {X 0,Y 361.963,Z 426.395,A -85,B 0,C 180,E1 -13154.621,E2 -13154.621} C_VEL
LIN {X 0,Y 361.961,Z 426.399,A -85,B 0,C 180,E1 -13158.099,E2 -13158.099} C_VEL
LIN {X 0,Y 361.893,Z 426.406,A -85,B 0,C 180,E1 -13161.653,E2 -13161.653} C_VEL
LIN {X 0,Y 361.93,Z 426.399,A -85,B 0,C 180,E1 -13165.29,E2 -13165.29} C_VEL
LIN {X 0,Y 361.91,Z 426.406,A -85,B 0,C 180,E1 -13167.779,E2 -13167.779} C_VEL
LIN {X 0,Y 361.839,Z 426.413,A -85,B 0,C 180,E1 -13171.63,E2 -13171.63} C_VEL
LIN {X 0,Y 361.876,Z 426.406,A -85,B 0,C 180,E1 -13175.345,E2 -13175.345} C_VEL
LIN {X 0,Y 361.872,Z 426.405,A -85,B 0,C 180,E1 -13179.027,E2 -13179.027} C_VEL
LIN {X 0,Y 361.839,Z 426.409,A -85,B 0,C 180,E1 -13182.829,E2 -13182.829} C_VEL
LIN {X 0,Y 361.823,Z 426.417,A -85,B 0,C 180,E1 -13185.946,E2 -13185.946} C_VEL
LIN {X 0,Y 361.838,Z 426.411,A -85,B 0,C 180,E1 -13189.245,E2 -13189.245} C_VEL
LIN {X 0,Y 361.867,Z 426.406,A -85,B 0,C 180,E1 -13192.777,E2 -13192.777} C_VEL
LIN {X 0,Y 361.859,Z 426.413,A -85,B 0,C 180,E1 -13195.72,E2 -13195.72} C_VEL
LIN {X 0,Y 361.879,Z 426.41,A -85,B 0,C 180,E1 -13199.673,E2 -13199.673} C_VEL
LIN {X 0,Y 361.958,Z 426.398,A -85,B 0,C 180,E1 -13203.476,E2 -13203.476} C_VEL
LIN {X 0,Y 361.894,Z 426.404,A -85,B 0,C 180,E1 -13207.145,E2 -13207.145} C_VEL
LIN {X 0,Y 361.925,Z 426.399,A -85,B 0,C 180,E1 -13210.725,E2 -13210.725} C_VEL
LIN {X 0,Y 361.954,Z 426.4,A -85,B 0,C 180,E1 -13214.25,E2 -13214.25} C_VEL
LIN {X 0,Y 365.948,Z 439.11,A -85,B 0,C 180,E1 -13215.369,E2 -13215.369} C_VEL
LIN {X 0,Y 367.769,Z 445.651,A -85,B 0,C 180,E1 -13216.039,E2 -13216.039} C_VEL
LIN {X 0,Y 367.373,Z 454.225,A -85,B 0,C 180,E1 -13216.884,E2 -13216.884} C_VEL
LIN {X 0,Y 366.476,Z 464.635,A -85,B 0,C 180,E1 -13218.121,E2 -13218.121} C_VEL
LIN {X 0,Y 365.555,Z 473.869,A -85,B 0,C 180,E1 -13219.476,E2 -13219.476} C_VEL
LIN {X 0,Y 364.779,Z 481.531,A -85,B 0,C 180,E1 -13220.854,E2 -13220.854} C_VEL
LIN {X 0,Y 363.941,Z 489.015,A -85,B 0,C 180,E1 -13222.511,E2 -13222.511} C_VEL
LIN {X 0,Y 363.411,Z 494.128,A -85,B 0,C 180,E1 -13223.894,E2 -13223.894} C_VEL
LIN {X 0,Y 362.911,Z 499.076,A -85,B 0,C 180,E1 -13225.558,E2 -13225.558} C_VEL
LIN {X 0,Y 362.47,Z 502.931,A -85,B 0,C 180,E1 -13227.222,E2 -13227.222} C_VEL
LIN {X 0,Y 362.1,Z 505.789,A -85,B 0,C 180,E1 -13228.888,E2 -13228.888} C_VEL
LIN {X 0,Y 361.966,Z 508.104,A -85,B 0,C 180,E1 -13231.113,E2 -13231.113} C_VEL
LIN {X 0,Y 361.886,Z 508.708,A -85,B 0,C 180,E1 -13232.226,E2 -13232.226} C_VEL
LIN {X 0,Y 361.765,Z 508.95,A -85,B 0,C 180,E1 -13233.341,E2 -13233.341} C_VEL
LIN {X 0,Y 362.044,Z 508.162,A -85,B 0,C 180,E1 -13235.57,E2 -13235.57} C_VEL
LIN {X 0,Y 362.358,Z 507.189,A -85,B 0,C 180,E1 -13236.683,E2 -13236.683} C_VEL
LIN {X 0,Y 362.514,Z 505.857,A -85,B 0,C 180,E1 -13237.8,E2 -13237.8} C_VEL
LIN {X 0,Y 362.948,Z 503.028,A -85,B 0,C 180,E1 -13239.474,E2 -13239.474} C_VEL
LIN {X 0,Y 363.546,Z 499.176,A -85,B 0,C 180,E1 -13241.147,E2 -13241.147} C_VEL
LIN {X 0,Y 364.233,Z 494.197,A -85,B 0,C 180,E1 -13242.821,E2 -13242.821} C_VEL
LIN {X 0,Y 364.943,Z 487.91,A -85,B 0,C 180,E1 -13244.499,E2 -13244.499} C_VEL
LIN {X 0,Y 365.987,Z 479.712,A -85,B 0,C 180,E1 -13246.229,E2 -13246.229} C_VEL
LIN {X 0,Y 366.926,Z 471.947,A -85,B 0,C 180,E1 -13247.558,E2 -13247.558} C_VEL
LIN {X 0,Y 367.875,Z 462.051,A -85,B 0,C 180,E1 -13248.952,E2 -13248.952} C_VEL
LIN {X 0,Y 368.792,Z 452.175,A -85,B 0,C 180,E1 -13250.061,E2 -13250.061} C_VEL
LIN {X 0,Y 369.043,Z 448.474,A -85,B 0,C 180,E1 -13250.428,E2 -13250.428} C_VEL
LIN {X 0,Y 365.906,Z 438.057,A -85,B 0,C 180,E1 -13251.557,E2 -13251.557} C_VEL
LIN {X 0,Y 361.891,Z 426.406,A -85,B 0,C 180,E1 -13252.648,E2 -13252.648} C_VEL
LIN {X 0,Y 361.959,Z 426.398,A -85,B 0,C 180,E1 -13256.525,E2 -13256.525} C_VEL
LIN {X 0,Y 361.879,Z 426.41,A -85,B 0,C 180,E1 -13260.328,E2 -13260.328} C_VEL
LIN {X 0,Y 361.859,Z 426.412,A -85,B 0,C 180,E1 -13264.28,E2 -13264.28} C_VEL
LIN {X 0,Y 361.868,Z 426.406,A -85,B 0,C 180,E1 -13267.223,E2 -13267.223} C_VEL
LIN {X 0,Y 361.855,Z 426.408,A -85,B 0,C 180,E1 -13269.527,E2 -13269.527} C_VEL
LIN {X 0,Y 361.182,Z 426.497,A -85,B 0,C 180,E1 -13270.456,E2 -13270.456} C_VEL
LIN {X 0,Y 358.301,Z 426.856,A -85,B 0,C 180,E1 -13271.967,E2 -13271.967} C_VEL
LIN {X 0,Y 355.871,Z 427.156,A -85,B 0,C 180,E1 -13273.19,E2 -13273.19} C_VEL
LIN {X 0,Y 354.843,Z 427.287,A -85,B 0,C 180,E1 -13274.136,E2 -13274.136} C_VEL
LIN {X 0,Y 354.767,Z 427.292,A -85,B 0,C 180,E1 -13274.457,E2 -13274.457} C_VEL
LIN {X 0,Y 354.799,Z 427.289,A -85,B 0,C 180,E1 -13277.663,E2 -13277.663} C_VEL
LIN {X 0,Y 354.819,Z 427.284,A -85,B 0,C 180,E1 -13280.666,E2 -13280.666} C_VEL
LIN {X 0,Y 354.826,Z 427.286,A -85,B 0,C 180,E1 -13284.301,E2 -13284.301} C_VEL
LIN {X 0,Y 354.792,Z 427.291,A -85,B 0,C 180,E1 -13287.667,E2 -13287.667} C_VEL
LIN {X 0,Y 354.873,Z 427.277,A -85,B 0,C 180,E1 -13290.621,E2 -13290.621} C_VEL
LIN {X 0,Y 354.903,Z 427.276,A -85,B 0,C 180,E1 -13294.173,E2 -13294.173} C_VEL
LIN {X 0,Y 354.821,Z 427.289,A -85,B 0,C 180,E1 -13297.893,E2 -13297.893} C_VEL
LIN {X 0,Y 354.927,Z 427.275,A -85,B 0,C 180,E1 -13301.891,E2 -13301.891} C_VEL
LIN {X 0,Y 354.957,Z 427.406,A -85,B 0,C 180,E1 -13303.408,E2 -13303.408} C_VEL
LIN {X 0,Y 358.017,Z 439.482,A -85,B 0,C 180,E1 -13304.45,E2 -13304.45} C_VEL
LIN {X 0,Y 358.9,Z 443.38,A -85,B 0,C 180,E1 -13304.831,E2 -13304.831} C_VEL
LIN {X 0,Y 358.242,Z 454.408,A -85,B 0,C 180,E1 -13305.949,E2 -13305.949} C_VEL
LIN {X 0,Y 357.643,Z 464.706,A -85,B 0,C 180,E1 -13307.228,E2 -13307.228} C_VEL
LIN {X 0,Y 356.945,Z 474.184,A -85,B 0,C 180,E1 -13308.644,E2 -13308.644} C_VEL
LIN {X 0,Y 356.27,Z 483.43,A -85,B 0,C 180,E1 -13310.348,E2 -13310.348} C_VEL
LIN {X 0,Y 355.728,Z 490.964,A -85,B 0,C 180,E1 -13312.05,E2 -13312.05} C_VEL
LIN {X 0,Y 355.364,Z 497.04,A -85,B 0,C 180,E1 -13313.755,E2 -13313.755} C_VEL
LIN {X 0,Y 354.894,Z 501.881,A -85,B 0,C 180,E1 -13315.457,E2 -13315.457} C_VEL
LIN {X 0,Y 354.777,Z 505.607,A -85,B 0,C 180,E1 -13317.161,E2 -13317.161} C_VEL
LIN {X 0,Y 354.79,Z 508.327,A -85,B 0,C 180,E1 -13318.865,E2 -13318.865} C_VEL
LIN {X 0,Y 354.929,Z 509.59,A -85,B 0,C 180,E1 -13320,E2 -13320} C_VEL
LIN {X 0,Y 354.999,Z 510.49,A -85,B 0,C 180,E1 -13321.134,E2 -13321.134} C_VEL
LIN {X 0,Y 355.139,Z 510.948,A -85,B 0,C 180,E1 -13322.268,E2 -13322.268} C_VEL
LIN {X 0,Y 355.479,Z 510.654,A -85,B 0,C 180,E1 -13324.536,E2 -13324.536} C_VEL
LIN {X 0,Y 355.728,Z 509.909,A -85,B 0,C 180,E1 -13325.669,E2 -13325.669} C_VEL
LIN {X 0,Y 356.567,Z 507.115,A -85,B 0,C 180,E1 -13327.93,E2 -13327.93} C_VEL
LIN {X 0,Y 357.369,Z 503.882,A -85,B 0,C 180,E1 -13329.623,E2 -13329.623} C_VEL
LIN {X 0,Y 358.328,Z 499.564,A -85,B 0,C 180,E1 -13331.311,E2 -13331.311} C_VEL
LIN {X 0,Y 359.545,Z 492.968,A -85,B 0,C 180,E1 -13333.278,E2 -13333.278} C_VEL
LIN {X 0,Y 360.881,Z 485.841,A -85,B 0,C 180,E1 -13334.954,E2 -13334.954} C_VEL
LIN {X 0,Y 362.34,Z 476.944,A -85,B 0,C 180,E1 -13336.624,E2 -13336.624} C_VEL
LIN {X 0,Y 363.683,Z 467.818,A -85,B 0,C 180,E1 -13338.011,E2 -13338.011} C_VEL
LIN {X 0,Y 365.245,Z 456.429,A -85,B 0,C 180,E1 -13339.393,E2 -13339.393} C_VEL
LIN {X 0,Y 365.35,Z 453.491,A -85,B 0,C 180,E1 -13339.736,E2 -13339.736} C_VEL
LIN {X 0,Y 362.353,Z 444.164,A -85,B 0,C 180,E1 -13341.071,E2 -13341.071} C_VEL
LIN {X 0,Y 358.625,Z 435.449,A -85,B 0,C 180,E1 -13342.314,E2 -13342.314} C_VEL
LIN {X 0,Y 355.051,Z 428.328,A -85,B 0,C 180,E1 -13343.321,E2 -13343.321} C_VEL
LIN {X 0,Y 354.848,Z 427.288,A -85,B 0,C 180,E1 -13343.462,E2 -13343.462} C_VEL
LIN {X 0,Y 354.887,Z 427.281,A -85,B 0,C 180,E1 -13347.096,E2 -13347.096} C_VEL
LIN {X 0,Y 354.857,Z 427.281,A -85,B 0,C 180,E1 -13349.678,E2 -13349.678} C_VEL
LIN {X 0,Y 354.809,Z 427.286,A -85,B 0,C 180,E1 -13353.702,E2 -13353.702} C_VEL
LIN {X 0,Y 354.801,Z 427.292,A -85,B 0,C 180,E1 -13356.459,E2 -13356.459} C_VEL
LIN {X 0,Y 354.826,Z 427.284,A -85,B 0,C 180,E1 -13359.423,E2 -13359.423} C_VEL
LIN {X 0,Y 354.843,Z 427.462,A -85,B 0,C 180,E1 -13363.464,E2 -13363.464} C_VEL
LIN {X 0,Y 356.812,Z 436.713,A -85,B 0,C 180,E1 -13367.418,E2 -13367.418} C_VEL
LIN {X 0,Y 358.322,Z 444.631,A -85,B 0,C 180,E1 -13370.566,E2 -13370.566} C_VEL
LIN {X 0,Y 359.011,Z 450.138,A -85,B 0,C 180,E1 -13372.637,E2 -13372.637} C_VEL
LIN {X 0,Y 357.581,Z 461.745,A -85,B 0,C 180,E1 -13376.611,E2 -13376.611} C_VEL
LIN {X 0,Y 356.4,Z 473.302,A -85,B 0,C 180,E1 -13380.463,E2 -13380.463} C_VEL
LIN {X 0,Y 355.417,Z 484.754,A -85,B 0,C 180,E1 -13384.213,E2 -13384.213} C_VEL
LIN {X 0,Y 354.713,Z 495.307,A -85,B 0,C 180,E1 -13387.579,E2 -13387.579} C_VEL
LIN {X 0,Y 357.485,Z 511.355,A -85,B 0,C 180,E1 -13388.789,E2 -13388.789} C_VEL
LIN {X 0,Y 358.456,Z 522.286,A -85,B 0,C 180,E1 -13389.664,E2 -13389.664} C_VEL
LIN {X 0,Y 358.576,Z 537.499,A -85,B 0,C 180,E1 -13391.026,E2 -13391.026} C_VEL
LIN {X 0,Y 358.173,Z 554.396,A -85,B 0,C 180,E1 -13392.735,E2 -13392.735} C_VEL
LIN {X 0,Y 356.855,Z 565.09,A -85,B 0,C 180,E1 -13393.995,E2 -13393.995} C_VEL
LIN {X 0,Y 355.742,Z 575.184,A -85,B 0,C 180,E1 -13395.476,E2 -13395.476} C_VEL
LIN {X 0,Y 354.84,Z 584.187,A -85,B 0,C 180,E1 -13397.125,E2 -13397.125} C_VEL
LIN {X 0,Y 354.23,Z 591.797,A -85,B 0,C 180,E1 -13398.846,E2 -13398.846} C_VEL
LIN {X 0,Y 353.889,Z 598.869,A -85,B 0,C 180,E1 -13400.858,E2 -13400.858} C_VEL
LIN {X 0,Y 353.863,Z 603.581,A -85,B 0,C 180,E1 -13402.582,E2 -13402.582} C_VEL
LIN {X 0,Y 353.975,Z 607.194,A -85,B 0,C 180,E1 -13404.302,E2 -13404.302} C_VEL
LIN {X 0,Y 354.143,Z 609.015,A -85,B 0,C 180,E1 -13405.447,E2 -13405.447} C_VEL
LIN {X 0,Y 354.239,Z 610.406,A -85,B 0,C 180,E1 -13406.588,E2 -13406.588} C_VEL
LIN {X 0,Y 354.308,Z 611.384,A -85,B 0,C 180,E1 -13407.726,E2 -13407.726} C_VEL
LIN {X 0,Y 354.639,Z 611.975,A -85,B 0,C 180,E1 -13408.864,E2 -13408.864} C_VEL
LIN {X 0,Y 354.699,Z 612.086,A -85,B 0,C 180,E1 -13410,E2 -13410} C_VEL
LIN {X 0,Y 354.649,Z 611.777,A -85,B 0,C 180,E1 -13411.135,E2 -13411.135} C_VEL
LIN {X 0,Y 354.286,Z 609.891,A -85,B 0,C 180,E1 -13413.412,E2 -13413.412} C_VEL
LIN {X 0,Y 354.144,Z 607.337,A -85,B 0,C 180,E1 -13415.123,E2 -13415.123} C_VEL
LIN {X 0,Y 353.964,Z 603.587,A -85,B 0,C 180,E1 -13416.9,E2 -13416.9} C_VEL
LIN {X 0,Y 353.92,Z 598.996,A -85,B 0,C 180,E1 -13418.565,E2 -13418.565} C_VEL
LIN {X 0,Y 354.12,Z 591.86,A -85,B 0,C 180,E1 -13420.578,E2 -13420.578} C_VEL
LIN {X 0,Y 354.617,Z 584.173,A -85,B 0,C 180,E1 -13422.301,E2 -13422.301} C_VEL
LIN {X 0,Y 355.24,Z 576.362,A -85,B 0,C 180,E1 -13423.733,E2 -13423.733} C_VEL
LIN {X 0,Y 355.793,Z 570.521,A -85,B 0,C 180,E1 -13424.648,E2 -13424.648} C_VEL
LIN {X 0,Y 356.826,Z 560.189,A -85,B 0,C 180,E1 -13426.006,E2 -13426.006} C_VEL
LIN {X 0,Y 357.697,Z 551.012,A -85,B 0,C 180,E1 -13426.993,E2 -13426.993} C_VEL
LIN {X 0,Y 357.488,Z 539.471,A -85,B 0,C 180,E1 -13428.037,E2 -13428.037} C_VEL
LIN {X 0,Y 356.954,Z 527.095,A -85,B 0,C 180,E1 -13428.924,E2 -13428.924} C_VEL
LIN {X 0,Y 355.903,Z 513.451,A -85,B 0,C 180,E1 -13429.652,E2 -13429.652} C_VEL
LIN {X 0,Y 354.305,Z 500.192,A -85,B 0,C 180,E1 -13430.16,E2 -13430.16} C_VEL
LIN {X 0,Y 354.851,Z 488.655,A -85,B 0,C 180,E1 -13433.865,E2 -13433.865} C_VEL
LIN {X 0,Y 355.699,Z 476.757,A -85,B 0,C 180,E1 -13437.692,E2 -13437.692} C_VEL
LIN {X 0,Y 356.731,Z 465.102,A -85,B 0,C 180,E1 -13441.472,E2 -13441.472} C_VEL
LIN {X 0,Y 357.905,Z 453.264,A -85,B 0,C 180,E1 -13445.4,E2 -13445.4} C_VEL
LIN {X 0,Y 358.505,Z 447.301,A -85,B 0,C 180,E1 -13447.424,E2 -13447.424} C_VEL
LIN {X 0,Y 357.705,Z 441.84,A -85,B 0,C 180,E1 -13449.428,E2 -13449.428} C_VEL
LIN {X 0,Y 356.113,Z 433.69,A -85,B 0,C 180,E1 -13452.582,E2 -13452.582} C_VEL
LIN {X 0,Y 354.808,Z 427.291,A -85,B 0,C 180,E1 -13455.253,E2 -13455.253} C_VEL
LIN {X 0,Y 354.789,Z 427.287,A -85,B 0,C 180,E1 -13459.179,E2 -13459.179} C_VEL
LIN {X 0,Y 354.813,Z 427.289,A -85,B 0,C 180,E1 -13462.401,E2 -13462.401} C_VEL
LIN {X 0,Y 354.813,Z 427.285,A -85,B 0,C 180,E1 -13464.941,E2 -13464.941} C_VEL
LIN {X 0,Y 354.794,Z 427.291,A -85,B 0,C 180,E1 -13468.405,E2 -13468.405} C_VEL
LIN {X 0,Y 354.847,Z 427.281,A -85,B 0,C 180,E1 -13471.619,E2 -13471.619} C_VEL
LIN {X 0,Y 354.9,Z 427.28,A -85,B 0,C 180,E1 -13474.173,E2 -13474.173} C_VEL
LIN {X 0,Y 354.835,Z 427.285,A -85,B 0,C 180,E1 -13477.894,E2 -13477.894} C_VEL
LIN {X 0,Y 354.923,Z 427.274,A -85,B 0,C 180,E1 -13481.891,E2 -13481.891} C_VEL
LIN {X 0,Y 354.944,Z 427.273,A -85,B 0,C 180,E1 -13485.981,E2 -13485.981} C_VEL
LIN {X 0,Y 354.981,Z 427.266,A -85,B 0,C 180,E1 -13489.736,E2 -13489.736} C_VEL
LIN {X 0,Y 355.115,Z 427.247,A -85,B 0,C 180,E1 -13493.18,E2 -13493.18} C_VEL
LIN {X 0,Y 355.248,Z 427.233,A -85,B 0,C 180,E1 -13497.733,E2 -13497.733} C_VEL
LIN {X 0,Y 355.399,Z 427.217,A -85,B 0,C 180,E1 -13500,E2 -13500} C_VEL
LIN {X 0,Y 355.245,Z 427.234,A -85,B 0,C 180,E1 -13502.268,E2 -13502.268} C_VEL
LIN {X 0,Y 355.14,Z 427.244,A -85,B 0,C 180,E1 -13506.819,E2 -13506.819} C_VEL
LIN {X 0,Y 355.016,Z 427.259,A -85,B 0,C 180,E1 -13509.113,E2 -13509.113} C_VEL
LIN {X 0,Y 354.923,Z 427.272,A -85,B 0,C 180,E1 -13512.581,E2 -13512.581} C_VEL
LIN {X 0,Y 354.891,Z 427.28,A -85,B 0,C 180,E1 -13516.096,E2 -13516.096} C_VEL
LIN {X 0,Y 354.908,Z 427.274,A -85,B 0,C 180,E1 -13518.472,E2 -13518.472} C_VEL
LIN {X 0,Y 354.836,Z 427.286,A -85,B 0,C 180,E1 -13522.106,E2 -13522.106} C_VEL
LIN {X 0,Y 354.901,Z 427.279,A -85,B 0,C 180,E1 -13525.828,E2 -13525.828} C_VEL
LIN {X 0,Y 354.819,Z 427.288,A -85,B 0,C 180,E1 -13529.682,E2 -13529.682} C_VEL
LIN {X 0,Y 354.807,Z 427.29,A -85,B 0,C 180,E1 -13533.702,E2 -13533.702} C_VEL
LIN {X 0,Y 354.801,Z 427.287,A -85,B 0,C 180,E1 -13536.46,E2 -13536.46} C_VEL
LIN {X 0,Y 354.825,Z 427.285,A -85,B 0,C 180,E1 -13539.424,E2 -13539.424} C_VEL
LIN {X 0,Y 354.791,Z 427.287,A -85,B 0,C 180,E1 -13542.868,E2 -13542.868} C_VEL
LIN {X 0,Y 354.771,Z 427.293,A -85,B 0,C 180,E1 -13546.104,E2 -13546.104} C_VEL
LIN {X 0,Y 354.791,Z 427.288,A -85,B 0,C 180,E1 -13549.18,E2 -13549.18} C_VEL
LIN {X 0,Y 354.811,Z 427.286,A -85,B 0,C 180,E1 -13552.403,E2 -13552.403} C_VEL
LIN {X 0,Y 354.815,Z 427.284,A -85,B 0,C 180,E1 -13554.941,E2 -13554.941} C_VEL
LIN {X 0,Y 354.818,Z 427.285,A -85,B 0,C 180,E1 -13558.4,E2 -13558.4} C_VEL
LIN {X 0,Y 354.857,Z 427.284,A -85,B 0,C 180,E1 -13561.62,E2 -13561.62} C_VEL
LIN {X 0,Y 354.903,Z 427.275,A -85,B 0,C 180,E1 -13564.173,E2 -13564.173} C_VEL
LIN {X 0,Y 354.838,Z 427.286,A -85,B 0,C 180,E1 -13567.894,E2 -13567.894} C_VEL
LIN {X 0,Y 354.926,Z 427.274,A -85,B 0,C 180,E1 -13571.892,E2 -13571.892} C_VEL
LIN {X 0,Y 354.897,Z 427.354,A -85,B 0,C 180,E1 -13573.905,E2 -13573.905} C_VEL
LIN {X 0,Y 358.504,Z 438.582,A -85,B 0,C 180,E1 -13574.888,E2 -13574.888} C_VEL
LIN {X 0,Y 360.903,Z 447.071,A -85,B 0,C 180,E1 -13575.768,E2 -13575.768} C_VEL
LIN {X 0,Y 360.972,Z 450.011,A -85,B 0,C 180,E1 -13576.058,E2 -13576.058} C_VEL
LIN {X 0,Y 360.093,Z 461.674,A -85,B 0,C 180,E1 -13577.345,E2 -13577.345} C_VEL
LIN {X 0,Y 359.093,Z 471.605,A -85,B 0,C 180,E1 -13578.714,E2 -13578.714} C_VEL
LIN {X 0,Y 358.196,Z 479.824,A -85,B 0,C 180,E1 -13580.115,E2 -13580.115} C_VEL
LIN {X 0,Y 357.246,Z 487.849,A -85,B 0,C 180,E1 -13581.8,E2 -13581.8} C_VEL
LIN {X 0,Y 356.556,Z 493.329,A -85,B 0,C 180,E1 -13583.208,E2 -13583.208} C_VEL
LIN {X 0,Y 356.121,Z 498.636,A -85,B 0,C 180,E1 -13584.905,E2 -13584.905} C_VEL
LIN {X 0,Y 355.567,Z 502.832,A -85,B 0,C 180,E1 -13586.601,E2 -13586.601} C_VEL
LIN {X 0,Y 355.276,Z 505.056,A -85,B 0,C 180,E1 -13587.733,E2 -13587.733} C_VEL
LIN {X 0,Y 355.079,Z 506.85,A -85,B 0,C 180,E1 -13588.866,E2 -13588.866} C_VEL
LIN {X 0,Y 354.95,Z 509.139,A -85,B 0,C 180,E1 -13591.135,E2 -13591.135} C_VEL
LIN {X 0,Y 354.861,Z 509.736,A -85,B 0,C 180,E1 -13592.27,E2 -13592.27} C_VEL
LIN {X 0,Y 354.742,Z 509.962,A -85,B 0,C 180,E1 -13593.408,E2 -13593.408} C_VEL
LIN {X 0,Y 355.043,Z 509.149,A -85,B 0,C 180,E1 -13595.68,E2 -13595.68} C_VEL
LIN {X 0,Y 355.373,Z 508.167,A -85,B 0,C 180,E1 -13596.815,E2 -13596.815} C_VEL
LIN {X 0,Y 355.542,Z 506.817,A -85,B 0,C 180,E1 -13597.954,E2 -13597.954} C_VEL
LIN {X 0,Y 356.017,Z 503.969,A -85,B 0,C 180,E1 -13599.66,E2 -13599.66} C_VEL
LIN {X 0,Y 356.641,Z 500.096,A -85,B 0,C 180,E1 -13601.365,E2 -13601.365} C_VEL
LIN {X 0,Y 357.365,Z 495.089,A -85,B 0,C 180,E1 -13603.071,E2 -13603.071} C_VEL
LIN {X 0,Y 358.105,Z 488.772,A -85,B 0,C 180,E1 -13604.782,E2 -13604.782} C_VEL
LIN {X 0,Y 359.222,Z 480.606,A -85,B 0,C 180,E1 -13606.53,E2 -13606.53} C_VEL
LIN {X 0,Y 360.211,Z 472.737,A -85,B 0,C 180,E1 -13607.897,E2 -13607.897} C_VEL
LIN {X 0,Y 361.206,Z 462.774,A -85,B 0,C 180,E1 -13609.316,E2 -13609.316} C_VEL
LIN {X 0,Y 362.285,Z 451.732,A -85,B 0,C 180,E1 -13610.553,E2 -13610.553} C_VEL
LIN {X 0,Y 362.093,Z 449.319,A -85,B 0,C 180,E1 -13610.82,E2 -13610.82} C_VEL
LIN {X 0,Y 359.026,Z 439.359,A -85,B 0,C 180,E1 -13611.933,E2 -13611.933} C_VEL
LIN {X 0,Y 354.844,Z 427.281,A -85,B 0,C 180,E1 -13613.102,E2 -13613.102} C_VEL
LIN {X 0,Y 354.893,Z 427.275,A -85,B 0,C 180,E1 -13616.982,E2 -13616.982} C_VEL
LIN {X 0,Y 354.858,Z 427.28,A -85,B 0,C 180,E1 -13619.679,E2 -13619.679} C_VEL
LIN {X 0,Y 354.81,Z 427.287,A -85,B 0,C 180,E1 -13623.702,E2 -13623.702} C_VEL
LIN {X 0,Y 354.803,Z 427.289,A -85,B 0,C 180,E1 -13626.459,E2 -13626.459} C_VEL
LIN {X 0,Y 354.819,Z 427.283,A -85,B 0,C 180,E1 -13629.51,E2 -13629.51} C_VEL
LIN {X 0,Y 354.792,Z 427.287,A -85,B 0,C 180,E1 -13632.867,E2 -13632.867} C_VEL
LIN {X 0,Y 354.767,Z 427.292,A -85,B 0,C 180,E1 -13634.457,E2 -13634.457} C_VEL
LIN {X 0,Y 354.114,Z 427.374,A -85,B 0,C 180,E1 -13635.403,E2 -13635.403} C_VEL
LIN {X 0,Y 351.248,Z 427.728,A -85,B 0,C 180,E1 -13636.942,E2 -13636.942} C_VEL
LIN {X 0,Y 348.822,Z 428.035,A -85,B 0,C 180,E1 -13638.188,E2 -13638.188} C_VEL
LIN {X 0,Y 347.799,Z 428.159,A -85,B 0,C 180,E1 -13639.153,E2 -13639.153} C_VEL
LIN {X 0,Y 347.727,Z 428.169,A -85,B 0,C 180,E1 -13639.479,E2 -13639.479} C_VEL
LIN {X 0,Y 347.766,Z 428.163,A -85,B 0,C 180,E1 -13642.679,E2 -13642.679} C_VEL
LIN {X 0,Y 347.752,Z 428.17,A -85,B 0,C 180,E1 -13645.956,E2 -13645.956} C_VEL
LIN {X 0,Y 347.768,Z 428.166,A -85,B 0,C 180,E1 -13649.654,E2 -13649.654} C_VEL
LIN {X 0,Y 347.856,Z 428.151,A -85,B 0,C 180,E1 -13652.745,E2 -13652.745} C_VEL
LIN {X 0,Y 347.789,Z 428.162,A -85,B 0,C 180,E1 -13656.162,E2 -13656.162} C_VEL
LIN {X 0,Y 347.816,Z 428.161,A -85,B 0,C 180,E1 -13659.909,E2 -13659.909} C_VEL
LIN {X 0,Y 347.885,Z 428.286,A -85,B 0,C 180,E1 -13663.193,E2 -13663.193} C_VEL
LIN {X 0,Y 351.022,Z 440.583,A -85,B 0,C 180,E1 -13664.274,E2 -13664.274} C_VEL
LIN {X 0,Y 351.945,Z 444.736,A -85,B 0,C 180,E1 -13664.691,E2 -13664.691} C_VEL
LIN {X 0,Y 351.164,Z 456.774,A -85,B 0,C 180,E1 -13665.956,E2 -13665.956} C_VEL
LIN {X 0,Y 350.592,Z 466.852,A -85,B 0,C 180,E1 -13667.261,E2 -13667.261} C_VEL
LIN {X 0,Y 349.839,Z 476.075,A -85,B 0,C 180,E1 -13668.704,E2 -13668.704} C_VEL
LIN {X 0,Y 349.234,Z 485.104,A -85,B 0,C 180,E1 -13670.43,E2 -13670.43} C_VEL
LIN {X 0,Y 348.677,Z 492.566,A -85,B 0,C 180,E1 -13672.18,E2 -13672.18} C_VEL
LIN {X 0,Y 348.179,Z 499.392,A -85,B 0,C 180,E1 -13674.207,E2 -13674.207} C_VEL
LIN {X 0,Y 347.924,Z 503.972,A -85,B 0,C 180,E1 -13675.946,E2 -13675.946} C_VEL
LIN {X 0,Y 347.744,Z 506.443,A -85,B 0,C 180,E1 -13677.104,E2 -13677.104} C_VEL
LIN {X 0,Y 347.765,Z 509.264,A -85,B 0,C 180,E1 -13678.842,E2 -13678.842} C_VEL
LIN {X 0,Y 347.91,Z 510.579,A -85,B 0,C 180,E1 -13680,E2 -13680} C_VEL
LIN {X 0,Y 347.984,Z 511.527,A -85,B 0,C 180,E1 -13681.157,E2 -13681.157} C_VEL
LIN {X 0,Y 348.132,Z 512.068,A -85,B 0,C 180,E1 -13682.314,E2 -13682.314} C_VEL
LIN {X 0,Y 348.52,Z 511.884,A -85,B 0,C 180,E1 -13684.626,E2 -13684.626} C_VEL
LIN {X 0,Y 348.811,Z 511.219,A -85,B 0,C 180,E1 -13685.782,E2 -13685.782} C_VEL
LIN {X 0,Y 349.19,Z 510.101,A -85,B 0,C 180,E1 -13686.936,E2 -13686.936} C_VEL
LIN {X 0,Y 349.696,Z 508.552,A -85,B 0,C 180,E1 -13688.087,E2 -13688.087} C_VEL
LIN {X 0,Y 350.549,Z 505.414,A -85,B 0,C 180,E1 -13689.812,E2 -13689.812} C_VEL
LIN {X 0,Y 351.678,Z 500.765,A -85,B 0,C 180,E1 -13691.697,E2 -13691.697} C_VEL
LIN {X 0,Y 352.886,Z 494.857,A -85,B 0,C 180,E1 -13693.533,E2 -13693.533} C_VEL
LIN {X 0,Y 354.301,Z 487.873,A -85,B 0,C 180,E1 -13695.238,E2 -13695.238} C_VEL
LIN {X 0,Y 355.857,Z 479.195,A -85,B 0,C 180,E1 -13696.936,E2 -13696.936} C_VEL
LIN {X 0,Y 357.558,Z 468.817,A -85,B 0,C 180,E1 -13698.569,E2 -13698.569} C_VEL
LIN {X 0,Y 359.168,Z 457.936,A -85,B 0,C 180,E1 -13699.917,E2 -13699.917} C_VEL
LIN {X 0,Y 359.253,Z 456.324,A -85,B 0,C 180,E1 -13700.112,E2 -13700.112} C_VEL
LIN {X 0,Y 356.238,Z 446.565,A -85,B 0,C 180,E1 -13701.592,E2 -13701.592} C_VEL
LIN {X 0,Y 351.69,Z 436.141,A -85,B 0,C 180,E1 -13703.183,E2 -13703.183} C_VEL
LIN {X 0,Y 348.35,Z 430.048,A -85,B 0,C 180,E1 -13704.153,E2 -13704.153} C_VEL
LIN {X 0,Y 347.818,Z 428.159,A -85,B 0,C 180,E1 -13704.391,E2 -13704.391} C_VEL
LIN {X 0,Y 347.814,Z 428.158,A -85,B 0,C 180,E1 -13707.694,E2 -13707.694} C_VEL
LIN {X 0,Y 347.767,Z 428.166,A -85,B 0,C 180,E1 -13710.346,E2 -13710.346} C_VEL
LIN {X 0,Y 347.747,Z 428.171,A -85,B 0,C 180,E1 -13714.464,E2 -13714.464} C_VEL
LIN {X 0,Y 347.776,Z 428.164,A -85,B 0,C 180,E1 -13717.988,E2 -13717.988} C_VEL
LIN {X 0,Y 347.753,Z 428.162,A -85,B 0,C 180,E1 -13721.83,E2 -13721.83} C_VEL
LIN {X 0,Y 347.755,Z 428.184,A -85,B 0,C 180,E1 -13722.9,E2 -13722.9} C_VEL
LIN {X 0,Y 349.399,Z 436.076,A -85,B 0,C 180,E1 -13726.396,E2 -13726.396} C_VEL
LIN {X 0,Y 350.693,Z 442.264,A -85,B 0,C 180,E1 -13728.978,E2 -13728.978} C_VEL
LIN {X 0,Y 351.917,Z 449.267,A -85,B 0,C 180,E1 -13731.75,E2 -13731.75} C_VEL
LIN {X 0,Y 351.849,Z 452.766,A -85,B 0,C 180,E1 -13733.033,E2 -13733.033} C_VEL
LIN {X 0,Y 350.298,Z 465.365,A -85,B 0,C 180,E1 -13737.42,E2 -13737.42} C_VEL
LIN {X 0,Y 349.137,Z 476.233,A -85,B 0,C 180,E1 -13741.111,E2 -13741.111} C_VEL
LIN {X 0,Y 348.164,Z 487.598,A -85,B 0,C 180,E1 -13744.918,E2 -13744.918} C_VEL
LIN {X 0,Y 347.81,Z 492.848,A -85,B 0,C 180,E1 -13746.676,E2 -13746.676} C_VEL
LIN {X 0,Y 348.525,Z 497.134,A -85,B 0,C 180,E1 -13747.006,E2 -13747.006} C_VEL
LIN {X 0,Y 351.066,Z 512.026,A -85,B 0,C 180,E1 -13748.237,E2 -13748.237} C_VEL
LIN {X 0,Y 351.96,Z 521.958,A -85,B 0,C 180,E1 -13749.103,E2 -13749.103} C_VEL
LIN {X 0,Y 352.005,Z 535.187,A -85,B 0,C 180,E1 -13750.325,E2 -13750.325} C_VEL
LIN {X 0,Y 351.532,Z 548.529,A -85,B 0,C 180,E1 -13751.797,E2 -13751.797} C_VEL
LIN {X 0,Y 351.071,Z 556.204,A -85,B 0,C 180,E1 -13752.675,E2 -13752.675} C_VEL
LIN {X 0,Y 349.787,Z 566.355,A -85,B 0,C 180,E1 -13753.962,E2 -13753.962} C_VEL
LIN {X 0,Y 348.592,Z 576.127,A -85,B 0,C 180,E1 -13755.499,E2 -13755.499} C_VEL
LIN {X 0,Y 347.885,Z 583.275,A -85,B 0,C 180,E1 -13756.863,E2 -13756.863} C_VEL
LIN {X 0,Y 347.201,Z 590.86,A -85,B 0,C 180,E1 -13758.617,E2 -13758.617} C_VEL
LIN {X 0,Y 346.833,Z 597.908,A -85,B 0,C 180,E1 -13760.671,E2 -13760.671} C_VEL
LIN {X 0,Y 346.798,Z 602.606,A -85,B 0,C 180,E1 -13762.43,E2 -13762.43} C_VEL
LIN {X 0,Y 346.902,Z 606.208,A -85,B 0,C 180,E1 -13764.186,E2 -13764.186} C_VEL
LIN {X 0,Y 347.08,Z 608.024,A -85,B 0,C 180,E1 -13765.354,E2 -13765.354} C_VEL
LIN {X 0,Y 347.189,Z 609.412,A -85,B 0,C 180,E1 -13766.518,E2 -13766.518} C_VEL
LIN {X 0,Y 347.263,Z 610.385,A -85,B 0,C 180,E1 -13767.68,E2 -13767.68} C_VEL
LIN {X 0,Y 347.606,Z 610.966,A -85,B 0,C 180,E1 -13768.841,E2 -13768.841} C_VEL
LIN {X 0,Y 347.674,Z 611.07,A -85,B 0,C 180,E1 -13770,E2 -13770} C_VEL
LIN {X 0,Y 347.618,Z 610.754,A -85,B 0,C 180,E1 -13771.158,E2 -13771.158} C_VEL
LIN {X 0,Y 347.308,Z 609.998,A -85,B 0,C 180,E1 -13772.319,E2 -13772.319} C_VEL
LIN {X 0,Y 347.237,Z 608.845,A -85,B 0,C 180,E1 -13773.481,E2 -13773.481} C_VEL
LIN {X 0,Y 347.084,Z 606.275,A -85,B 0,C 180,E1 -13775.228,E2 -13775.228} C_VEL
LIN {X 0,Y 346.901,Z 602.645,A -85,B 0,C 180,E1 -13776.982,E2 -13776.982} C_VEL
LIN {X 0,Y 346.845,Z 597.893,A -85,B 0,C 180,E1 -13778.741,E2 -13778.741} C_VEL
LIN {X 0,Y 347.038,Z 591.892,A -85,B 0,C 180,E1 -13780.501,E2 -13780.501} C_VEL
LIN {X 0,Y 347.509,Z 584.42,A -85,B 0,C 180,E1 -13782.26,E2 -13782.26} C_VEL
LIN {X 0,Y 348.164,Z 576.865,A -85,B 0,C 180,E1 -13783.72,E2 -13783.72} C_VEL
LIN {X 0,Y 348.565,Z 571.726,A -85,B 0,C 180,E1 -13784.577,E2 -13784.577} C_VEL
LIN {X 0,Y 349.61,Z 562.457,A -85,B 0,C 180,E1 -13785.896,E2 -13785.896} C_VEL
LIN {X 0,Y 350.696,Z 551.176,A -85,B 0,C 180,E1 -13787.193,E2 -13787.193} C_VEL
LIN {X 0,Y 350.52,Z 539.917,A -85,B 0,C 180,E1 -13788.257,E2 -13788.257} C_VEL
LIN {X 0,Y 350.04,Z 526.934,A -85,B 0,C 180,E1 -13789.228,E2 -13789.228} C_VEL
LIN {X 0,Y 349.066,Z 514.164,A -85,B 0,C 180,E1 -13789.954,E2 -13789.954} C_VEL
LIN {X 0,Y 347.321,Z 499.926,A -85,B 0,C 180,E1 -13790.529,E2 -13790.529} C_VEL
LIN {X 0,Y 347.293,Z 499.056,A -85,B 0,C 180,E1 -13790.586,E2 -13790.586} C_VEL
LIN {X 0,Y 347.929,Z 486.772,A -85,B 0,C 180,E1 -13794.635,E2 -13794.635} C_VEL
LIN {X 0,Y 348.74,Z 475.776,A -85,B 0,C 180,E1 -13798.267,E2 -13798.267} C_VEL
LIN {X 0,Y 349.692,Z 466.043,A -85,B 0,C 180,E1 -13801.503,E2 -13801.503} C_VEL
LIN {X 0,Y 350.902,Z 454.24,A -85,B 0,C 180,E1 -13805.508,E2 -13805.508} C_VEL
LIN {X 0,Y 351.509,Z 448.294,A -85,B 0,C 180,E1 -13807.576,E2 -13807.576} C_VEL
LIN {X 0,Y 350.553,Z 442.108,A -85,B 0,C 180,E1 -13809.907,E2 -13809.907} C_VEL
LIN {X 0,Y 348.782,Z 433.143,A -85,B 0,C 180,E1 -13813.497,E2 -13813.497} C_VEL
LIN {X 0,Y 347.757,Z 428.168,A -85,B 0,C 180,E1 -13815.694,E2 -13815.694} C_VEL
LIN {X 0,Y 347.751,Z 428.17,A -85,B 0,C 180,E1 -13818.397,E2 -13818.397} C_VEL
LIN {X 0,Y 347.777,Z 428.165,A -85,B 0,C 180,E1 -13822.01,E2 -13822.01} C_VEL
LIN {X 0,Y 347.745,Z 428.166,A -85,B 0,C 180,E1 -13825.536,E2 -13825.536} C_VEL
LIN {X 0,Y 347.745,Z 428.17,A -85,B 0,C 180,E1 -13828.3,E2 -13828.3} C_VEL
LIN {X 0,Y 347.779,Z 428.161,A -85,B 0,C 180,E1 -13830.988,E2 -13830.988} C_VEL
LIN {X 0,Y 347.831,Z 428.155,A -85,B 0,C 180,E1 -13833.608,E2 -13833.608} C_VEL
LIN {X 0,Y 347.789,Z 428.166,A -85,B 0,C 180,E1 -13836.162,E2 -13836.162} C_VEL
LIN {X 0,Y 347.818,Z 428.16,A -85,B 0,C 180,E1 -13839.91,E2 -13839.91} C_VEL
LIN {X 0,Y 347.867,Z 428.154,A -85,B 0,C 180,E1 -13842.359,E2 -13842.359} C_VEL
LIN {X 0,Y 347.898,Z 428.151,A -85,B 0,C 180,E1 -13845.971,E2 -13845.971} C_VEL
LIN {X 0,Y 347.932,Z 428.143,A -85,B 0,C 180,E1 -13849.526,E2 -13849.526} C_VEL
LIN {X 0,Y 348.083,Z 428.123,A -85,B 0,C 180,E1 -13853.042,E2 -13853.042} C_VEL
LIN {X 0,Y 348.21,Z 428.11,A -85,B 0,C 180,E1 -13857.687,E2 -13857.687} C_VEL
LIN {X 0,Y 348.369,Z 428.093,A -85,B 0,C 180,E1 -13860,E2 -13860} C_VEL
LIN {X 0,Y 348.207,Z 428.111,A -85,B 0,C 180,E1 -13862.314,E2 -13862.314} C_VEL
LIN {X 0,Y 348.108,Z 428.119,A -85,B 0,C 180,E1 -13866.958,E2 -13866.958} C_VEL
LIN {X 0,Y 347.969,Z 428.138,A -85,B 0,C 180,E1 -13869.299,E2 -13869.299} C_VEL
LIN {X 0,Y 347.892,Z 428.146,A -85,B 0,C 180,E1 -13872.84,E2 -13872.84} C_VEL
LIN {X 0,Y 347.841,Z 428.155,A -85,B 0,C 180,E1 -13876.432,E2 -13876.432} C_VEL
LIN {X 0,Y 347.857,Z 428.151,A -85,B 0,C 180,E1 -13878.86,E2 -13878.86} C_VEL
LIN {X 0,Y 347.776,Z 428.161,A -85,B 0,C 180,E1 -13882.58,E2 -13882.58} C_VEL
LIN {X 0,Y 347.813,Z 428.156,A -85,B 0,C 180,E1 -13885.109,E2 -13885.109} C_VEL
LIN {X 0,Y 347.809,Z 428.161,A -85,B 0,C 180,E1 -13887.694,E2 -13887.694} C_VEL
LIN {X 0,Y 347.75,Z 428.166,A -85,B 0,C 180,E1 -13890.348,E2 -13890.348} C_VEL
LIN {X 0,Y 347.749,Z 428.168,A -85,B 0,C 180,E1 -13894.044,E2 -13894.044} C_VEL
LIN {X 0,Y 347.764,Z 428.164,A -85,B 0,C 180,E1 -13897.321,E2 -13897.321} C_VEL
LIN {X 0,Y 347.734,Z 428.168,A -85,B 0,C 180,E1 -13900.297,E2 -13900.297} C_VEL
LIN {X 0,Y 347.726,Z 428.169,A -85,B 0,C 180,E1 -13903.408,E2 -13903.408} C_VEL
LIN {X 0,Y 347.728,Z 428.167,A -85,B 0,C 180,E1 -13906.686,E2 -13906.686} C_VEL
LIN {X 0,Y 347.75,Z 428.167,A -85,B 0,C 180,E1 -13910.173,E2 -13910.173} C_VEL
LIN {X 0,Y 347.765,Z 428.162,A -85,B 0,C 180,E1 -13912.68,E2 -13912.68} C_VEL
LIN {X 0,Y 347.751,Z 428.168,A -85,B 0,C 180,E1 -13915.957,E2 -13915.957} C_VEL
LIN {X 0,Y 347.773,Z 428.167,A -85,B 0,C 180,E1 -13919.655,E2 -13919.655} C_VEL
LIN {X 0,Y 347.836,Z 428.159,A -85,B 0,C 180,E1 -13923.608,E2 -13923.608} C_VEL
LIN {X 0,Y 347.792,Z 428.161,A -85,B 0,C 180,E1 -13926.162,E2 -13926.162} C_VEL
LIN {X 0,Y 347.821,Z 428.16,A -85,B 0,C 180,E1 -13929.91,E2 -13929.91} C_VEL
LIN {X 0,Y 347.866,Z 428.151,A -85,B 0,C 180,E1 -13932.966,E2 -13932.966} C_VEL
LIN {X 0,Y 347.873,Z 428.154,A -85,B 0,C 180,E1 -13933.495,E2 -13933.495} C_VEL
LIN {X 0,Y 351.688,Z 440.156,A -85,B 0,C 180,E1 -13934.592,E2 -13934.592} C_VEL
LIN {X 0,Y 354.32,Z 449.953,A -85,B 0,C 180,E1 -13935.645,E2 -13935.645} C_VEL
LIN {X 0,Y 353.499,Z 460.447,A -85,B 0,C 180,E1 -13936.784,E2 -13936.784} C_VEL
LIN {X 0,Y 352.438,Z 470.841,A -85,B 0,C 180,E1 -13938.187,E2 -13938.187} C_VEL
LIN {X 0,Y 351.427,Z 479.516,A -85,B 0,C 180,E1 -13939.631,E2 -13939.631} C_VEL
LIN {X 0,Y 350.498,Z 487.804,A -85,B 0,C 180,E1 -13941.351,E2 -13941.351} C_VEL
LIN {X 0,Y 349.598,Z 494.463,A -85,B 0,C 180,E1 -13943.072,E2 -13943.072} C_VEL
LIN {X 0,Y 349.149,Z 499.744,A -85,B 0,C 180,E1 -13944.803,E2 -13944.803} C_VEL
LIN {X 0,Y 348.562,Z 503.919,A -85,B 0,C 180,E1 -13946.532,E2 -13946.532} C_VEL
LIN {X 0,Y 348.26,Z 506.133,A -85,B 0,C 180,E1 -13947.687,E2 -13947.687} C_VEL
LIN {X 0,Y 348.057,Z 507.908,A -85,B 0,C 180,E1 -13948.843,E2 -13948.843} C_VEL
LIN {X 0,Y 347.932,Z 510.175,A -85,B 0,C 180,E1 -13951.158,E2 -13951.158} C_VEL
LIN {X 0,Y 347.837,Z 510.763,A -85,B 0,C 180,E1 -13952.316,E2 -13952.316} C_VEL
LIN {X 0,Y 347.719,Z 510.972,A -85,B 0,C 180,E1 -13953.477,E2 -13953.477} C_VEL
LIN {X 0,Y 348.044,Z 510.137,A -85,B 0,C 180,E1 -13955.795,E2 -13955.795} C_VEL
LIN {X 0,Y 348.389,Z 509.144,A -85,B 0,C 180,E1 -13956.952,E2 -13956.952} C_VEL
LIN {X 0,Y 348.574,Z 507.776,A -85,B 0,C 180,E1 -13958.114,E2 -13958.114} C_VEL
LIN {X 0,Y 349.089,Z 504.909,A -85,B 0,C 180,E1 -13959.854,E2 -13959.854} C_VEL
LIN {X 0,Y 349.743,Z 501.014,A -85,B 0,C 180,E1 -13961.593,E2 -13961.593} C_VEL
LIN {X 0,Y 350.507,Z 495.978,A -85,B 0,C 180,E1 -13963.332,E2 -13963.332} C_VEL
LIN {X 0,Y 351.281,Z 489.634,A -85,B 0,C 180,E1 -13965.076,E2 -13965.076} C_VEL
LIN {X 0,Y 352.471,Z 481.487,A -85,B 0,C 180,E1 -13966.845,E2 -13966.845} C_VEL
LIN {X 0,Y 353.51,Z 473.529,A -85,B 0,C 180,E1 -13968.248,E2 -13968.248} C_VEL
LIN {X 0,Y 354.544,Z 463.497,A -85,B 0,C 180,E1 -13969.694,E2 -13969.694} C_VEL
LIN {X 0,Y 355.684,Z 452.331,A -85,B 0,C 180,E1 -13970.959,E2 -13970.959} C_VEL
LIN {X 0,Y 352.337,Z 441.149,A -85,B 0,C 180,E1 -13972.271,E2 -13972.271} C_VEL
LIN {X 0,Y 348.877,Z 431.47,A -85,B 0,C 180,E1 -13973.248,E2 -13973.248} C_VEL
LIN {X 0,Y 347.786,Z 428.16,A -85,B 0,C 180,E1 -13973.55,E2 -13973.55} C_VEL
LIN {X 0,Y 347.856,Z 428.151,A -85,B 0,C 180,E1 -13977.255,E2 -13977.255} C_VEL
LIN {X 0,Y 347.768,Z 428.168,A -85,B 0,C 180,E1 -13980.347,E2 -13980.347} C_VEL
LIN {X 0,Y 347.748,Z 428.168,A -85,B 0,C 180,E1 -13984.464,E2 -13984.464} C_VEL
LIN {X 0,Y 347.778,Z 428.166,A -85,B 0,C 180,E1 -13987.989,E2 -13987.989} C_VEL
LIN {X 0,Y 347.755,Z 428.167,A -85,B 0,C 180,E1 -13991.83,E2 -13991.83} C_VEL
LIN {X 0,Y 347.71,Z 428.169,A -85,B 0,C 180,E1 -13995.027,E2 -13995.027} C_VEL
LIN {X 0,Y 347.754,Z 428.166,A -85,B 0,C 180,E1 -13998.397,E2 -13998.397} C_VEL
LIN {X 0,Y 347.727,Z 428.169,A -85,B 0,C 180,E1 -13999.479,E2 -13999.479} C_VEL
LIN {X 0,Y 347.08,Z 428.254,A -85,B 0,C 180,E1 -14000.445,E2 -14000.445} C_VEL
LIN {X 0,Y 344.214,Z 428.611,A -85,B 0,C 180,E1 -14002.016,E2 -14002.016} C_VEL
LIN {X 0,Y 341.791,Z 428.907,A -85,B 0,C 180,E1 -14003.288,E2 -14003.288} C_VEL
LIN {X 0,Y 340.78,Z 429.035,A -85,B 0,C 180,E1 -14004.273,E2 -14004.273} C_VEL
LIN {X 0,Y 340.715,Z 429.04,A -85,B 0,C 180,E1 -14004.606,E2 -14004.606} C_VEL
LIN {X 0,Y 340.695,Z 429.047,A -85,B 0,C 180,E1 -14007.755,E2 -14007.755} C_VEL
LIN {X 0,Y 340.778,Z 429.035,A -85,B 0,C 180,E1 -14010.332,E2 -14010.332} C_VEL
LIN {X 0,Y 340.809,Z 429.029,A -85,B 0,C 180,E1 -14013.02,E2 -14013.02} C_VEL
LIN {X 0,Y 340.758,Z 429.039,A -85,B 0,C 180,E1 -14015.638,E2 -14015.638} C_VEL
LIN {X 0,Y 340.742,Z 429.04,A -85,B 0,C 180,E1 -14019.474,E2 -14019.474} C_VEL
LIN {X 0,Y 340.847,Z 429.025,A -85,B 0,C 180,E1 -14022.951,E2 -14022.951} C_VEL
LIN {X 0,Y 344.267,Z 442.726,A -85,B 0,C 180,E1 -14024.221,E2 -14024.221} C_VEL
LIN {X 0,Y 344.94,Z 445.646,A -85,B 0,C 180,E1 -14024.519,E2 -14024.519} C_VEL
LIN {X 0,Y 344.144,Z 457.691,A -85,B 0,C 180,E1 -14025.814,E2 -14025.814} C_VEL
LIN {X 0,Y 343.509,Z 468.782,A -85,B 0,C 180,E1 -14027.294,E2 -14027.294} C_VEL
LIN {X 0,Y 342.62,Z 479.509,A -85,B 0,C 180,E1 -14029.062,E2 -14029.062} C_VEL
LIN {X 0,Y 342.053,Z 487.897,A -85,B 0,C 180,E1 -14030.778,E2 -14030.778} C_VEL
LIN {X 0,Y 341.517,Z 495.186,A -85,B 0,C 180,E1 -14032.61,E2 -14032.61} C_VEL
LIN {X 0,Y 341.128,Z 501.709,A -85,B 0,C 180,E1 -14034.68,E2 -14034.68} C_VEL
LIN {X 0,Y 340.627,Z 506.052,A -85,B 0,C 180,E1 -14036.451,E2 -14036.451} C_VEL
LIN {X 0,Y 340.817,Z 508.306,A -85,B 0,C 180,E1 -14037.636,E2 -14037.636} C_VEL
LIN {X 0,Y 340.74,Z 510.177,A -85,B 0,C 180,E1 -14038.818,E2 -14038.818} C_VEL
LIN {X 0,Y 340.889,Z 511.563,A -85,B 0,C 180,E1 -14040,E2 -14040} C_VEL
LIN {X 0,Y 341.123,Z 513.176,A -85,B 0,C 180,E1 -14042.361,E2 -14042.361} C_VEL
LIN {X 0,Y 341.319,Z 513.362,A -85,B 0,C 180,E1 -14043.541,E2 -14043.541} C_VEL
LIN {X 0,Y 341.89,Z 512.513,A -85,B 0,C 180,E1 -14045.899,E2 -14045.899} C_VEL
LIN {X 0,Y 342.284,Z 511.489,A -85,B 0,C 180,E1 -14047.076,E2 -14047.076} C_VEL
LIN {X 0,Y 343.381,Z 508.126,A -85,B 0,C 180,E1 -14049.424,E2 -14049.424} C_VEL
LIN {X 0,Y 344.559,Z 504.037,A -85,B 0,C 180,E1 -14051.342,E2 -14051.342} C_VEL
LIN {X 0,Y 345.596,Z 499.634,A -85,B 0,C 180,E1 -14052.926,E2 -14052.926} C_VEL
LIN {X 0,Y 346.973,Z 493.515,A -85,B 0,C 180,E1 -14054.666,E2 -14054.666} C_VEL
LIN {X 0,Y 348.6,Z 485.984,A -85,B 0,C 180,E1 -14056.394,E2 -14056.394} C_VEL
LIN {X 0,Y 350.026,Z 478.362,A -85,B 0,C 180,E1 -14057.83,E2 -14057.83} C_VEL
LIN {X 0,Y 351.627,Z 469.08,A -85,B 0,C 180,E1 -14059.256,E2 -14059.256} C_VEL
LIN {X 0,Y 353.122,Z 459.41,A -85,B 0,C 180,E1 -14060.477,E2 -14060.477} C_VEL
LIN {X 0,Y 351.355,Z 452.595,A -85,B 0,C 180,E1 -14061.571,E2 -14061.571} C_VEL
LIN {X 0,Y 348.076,Z 444.043,A -85,B 0,C 180,E1 -14062.964,E2 -14062.964} C_VEL
LIN {X 0,Y 343.906,Z 435.447,A -85,B 0,C 180,E1 -14064.397,E2 -14064.397} C_VEL
LIN {X 0,Y 342.783,Z 433.145,A -85,B 0,C 180,E1 -14064.782,E2 -14064.782} C_VEL
LIN {X 0,Y 341.536,Z 431.46,A -85,B 0,C 180,E1 -14065.12,E2 -14065.12} C_VEL
LIN {X 0,Y 340.758,Z 429.039,A -85,B 0,C 180,E1 -14065.488,E2 -14065.488} C_VEL
LIN {X 0,Y 340.744,Z 429.039,A -85,B 0,C 180,E1 -14068.319,E2 -14068.319} C_VEL
LIN {X 0,Y 340.706,Z 429.045,A -85,B 0,C 180,E1 -14071.044,E2 -14071.044} C_VEL
LIN {X 0,Y 340.721,Z 429.042,A -85,B 0,C 180,E1 -14075.279,E2 -14075.279} C_VEL
LIN {X 0,Y 340.712,Z 429.047,A -85,B 0,C 180,E1 -14078.386,E2 -14078.386} C_VEL
LIN {X 0,Y 340.735,Z 429.115,A -85,B 0,C 180,E1 -14082.419,E2 -14082.419} C_VEL
LIN {X 0,Y 342.305,Z 436.822,A -85,B 0,C 180,E1 -14085.939,E2 -14085.939} C_VEL
LIN {X 0,Y 343.867,Z 444.342,A -85,B 0,C 180,E1 -14089.154,E2 -14089.154} C_VEL
LIN {X 0,Y 344.937,Z 450.384,A -85,B 0,C 180,E1 -14091.589,E2 -14091.589} C_VEL
LIN {X 0,Y 344.987,Z 453.084,A -85,B 0,C 180,E1 -14092.608,E2 -14092.608} C_VEL
LIN {X 0,Y 343.386,Z 465.503,A -85,B 0,C 180,E1 -14097.049,E2 -14097.049} C_VEL
LIN {X 0,Y 342.069,Z 477.223,A -85,B 0,C 180,E1 -14101.13,E2 -14101.13} C_VEL
LIN {X 0,Y 341.058,Z 488.628,A -85,B 0,C 180,E1 -14105.051,E2 -14105.051} C_VEL
LIN {X 0,Y 340.913,Z 490.813,A -85,B 0,C 180,E1 -14105.731,E2 -14105.731} C_VEL
LIN {X 0,Y 341.782,Z 495.234,A -85,B 0,C 180,E1 -14106.105,E2 -14106.105} C_VEL
LIN {X 0,Y 344.274,Z 509.43,A -85,B 0,C 180,E1 -14107.363,E2 -14107.363} C_VEL
LIN {X 0,Y 345.506,Z 521.962,A -85,B 0,C 180,E1 -14108.522,E2 -14108.522} C_VEL
LIN {X 0,Y 345.412,Z 536.083,A -85,B 0,C 180,E1 -14109.923,E2 -14109.923} C_VEL
LIN {X 0,Y 344.798,Z 549.07,A -85,B 0,C 180,E1 -14111.428,E2 -14111.428} C_VEL
LIN {X 0,Y 344.125,Z 556.834,A -85,B 0,C 180,E1 -14112.468,E2 -14112.468} C_VEL
LIN {X 0,Y 342.664,Z 567.479,A -85,B 0,C 180,E1 -14113.925,E2 -14113.925} C_VEL
LIN {X 0,Y 341.574,Z 575.969,A -85,B 0,C 180,E1 -14115.329,E2 -14115.329} C_VEL
LIN {X 0,Y 340.737,Z 583.746,A -85,B 0,C 180,E1 -14116.886,E2 -14116.886} C_VEL
LIN {X 0,Y 340.101,Z 591.061,A -85,B 0,C 180,E1 -14118.678,E2 -14118.678} C_VEL
LIN {X 0,Y 339.757,Z 596.944,A -85,B 0,C 180,E1 -14120.474,E2 -14120.474} C_VEL
LIN {X 0,Y 339.728,Z 601.631,A -85,B 0,C 180,E1 -14122.272,E2 -14122.272} C_VEL
LIN {X 0,Y 339.828,Z 605.221,A -85,B 0,C 180,E1 -14124.064,E2 -14124.064} C_VEL
LIN {X 0,Y 340.018,Z 607.034,A -85,B 0,C 180,E1 -14125.257,E2 -14125.257} C_VEL
LIN {X 0,Y 340.141,Z 608.418,A -85,B 0,C 180,E1 -14126.446,E2 -14126.446} C_VEL
LIN {X 0,Y 340.218,Z 609.386,A -85,B 0,C 180,E1 -14127.632,E2 -14127.632} C_VEL
LIN {X 0,Y 340.573,Z 609.956,A -85,B 0,C 180,E1 -14128.817,E2 -14128.817} C_VEL
LIN {X 0,Y 340.649,Z 610.055,A -85,B 0,C 180,E1 -14130,E2 -14130} C_VEL
LIN {X 0,Y 340.586,Z 609.731,A -85,B 0,C 180,E1 -14131.182,E2 -14131.182} C_VEL
LIN {X 0,Y 340.265,Z 608.966,A -85,B 0,C 180,E1 -14132.367,E2 -14132.367} C_VEL
LIN {X 0,Y 340.188,Z 607.797,A -85,B 0,C 180,E1 -14133.553,E2 -14133.553} C_VEL
LIN {X 0,Y 340.024,Z 605.212,A -85,B 0,C 180,E1 -14135.337,E2 -14135.337} C_VEL
LIN {X 0,Y 339.818,Z 601.562,A -85,B 0,C 180,E1 -14137.128,E2 -14137.128} C_VEL
LIN {X 0,Y 339.792,Z 596.792,A -85,B 0,C 180,E1 -14138.924,E2 -14138.924} C_VEL
LIN {X 0,Y 339.976,Z 590.76,A -85,B 0,C 180,E1 -14140.722,E2 -14140.722} C_VEL
LIN {X 0,Y 340.503,Z 583.269,A -85,B 0,C 180,E1 -14142.516,E2 -14142.516} C_VEL
LIN {X 0,Y 341.081,Z 575.67,A -85,B 0,C 180,E1 -14144.011,E2 -14144.011} C_VEL
LIN {X 0,Y 342.336,Z 565.562,A -85,B 0,C 180,E1 -14145.631,E2 -14145.631} C_VEL
LIN {X 0,Y 343.3,Z 555.26,A -85,B 0,C 180,E1 -14146.961,E2 -14146.961} C_VEL
LIN {X 0,Y 343.67,Z 549.858,A -85,B 0,C 180,E1 -14147.556,E2 -14147.556} C_VEL
LIN {X 0,Y 343.488,Z 538.525,A -85,B 0,C 180,E1 -14148.644,E2 -14148.644} C_VEL
LIN {X 0,Y 343.102,Z 526.436,A -85,B 0,C 180,E1 -14149.567,E2 -14149.567} C_VEL
LIN {X 0,Y 342.104,Z 513.438,A -85,B 0,C 180,E1 -14150.335,E2 -14150.335} C_VEL
LIN {X 0,Y 340.402,Z 499.867,A -85,B 0,C 180,E1 -14150.91,E2 -14150.91} C_VEL
LIN {X 0,Y 340.228,Z 497.956,A -85,B 0,C 180,E1 -14151.03,E2 -14151.03} C_VEL
LIN {X 0,Y 340.971,Z 485.583,A -85,B 0,C 180,E1 -14155.206,E2 -14155.206} C_VEL
LIN {X 0,Y 341.83,Z 474.72,A -85,B 0,C 180,E1 -14158.892,E2 -14158.892} C_VEL
LIN {X 0,Y 342.792,Z 464.997,A -85,B 0,C 180,E1 -14162.212,E2 -14162.212} C_VEL
LIN {X 0,Y 344.169,Z 453.24,A -85,B 0,C 180,E1 -14166.312,E2 -14166.312} C_VEL
LIN {X 0,Y 344.512,Z 449.276,A -85,B 0,C 180,E1 -14167.734,E2 -14167.734} C_VEL
LIN {X 0,Y 343.236,Z 441.529,A -85,B 0,C 180,E1 -14170.747,E2 -14170.747} C_VEL
LIN {X 0,Y 341.47,Z 432.703,A -85,B 0,C 180,E1 -14174.409,E2 -14174.409} C_VEL
LIN {X 0,Y 340.694,Z 429.049,A -85,B 0,C 180,E1 -14176.054,E2 -14176.054} C_VEL
LIN {X 0,Y 340.689,Z 429.047,A -85,B 0,C 180,E1 -14179.753,E2 -14179.753} C_VEL
LIN {X 0,Y 340.707,Z 429.042,A -85,B 0,C 180,E1 -14183.259,E2 -14183.259} C_VEL
LIN {X 0,Y 340.695,Z 429.049,A -85,B 0,C 180,E1 -14186.154,E2 -14186.154} C_VEL
LIN {X 0,Y 340.741,Z 429.042,A -85,B 0,C 180,E1 -14190.329,E2 -14190.329} C_VEL
LIN {X 0,Y 340.803,Z 429.03,A -85,B 0,C 180,E1 -14193.02,E2 -14193.02} C_VEL
LIN {X 0,Y 340.756,Z 429.037,A -85,B 0,C 180,E1 -14195.638,E2 -14195.638} C_VEL
LIN {X 0,Y 340.756,Z 429.036,A -85,B 0,C 180,E1 -14199.475,E2 -14199.475} C_VEL
LIN {X 0,Y 340.859,Z 429.028,A -85,B 0,C 180,E1 -14201.984,E2 -14201.984} C_VEL
LIN {X 0,Y 340.87,Z 429.024,A -85,B 0,C 180,E1 -14205.705,E2 -14205.705} C_VEL
LIN {X 0,Y 340.875,Z 429.021,A -85,B 0,C 180,E1 -14209.306,E2 -14209.306} C_VEL
LIN {X 0,Y 341.05,Z 428.999,A -85,B 0,C 180,E1 -14212.898,E2 -14212.898} C_VEL
LIN {X 0,Y 341.172,Z 428.986,A -85,B 0,C 180,E1 -14217.639,E2 -14217.639} C_VEL
LIN {X 0,Y 341.317,Z 428.971,A -85,B 0,C 180,E1 -14220,E2 -14220} C_VEL
LIN {X 0,Y 341.169,Z 428.987,A -85,B 0,C 180,E1 -14222.361,E2 -14222.361} C_VEL
LIN {X 0,Y 341.077,Z 428.995,A -85,B 0,C 180,E1 -14227.102,E2 -14227.102} C_VEL
LIN {X 0,Y 340.872,Z 429.021,A -85,B 0,C 180,E1 -14230.694,E2 -14230.694} C_VEL
LIN {X 0,Y 340.864,Z 429.025,A -85,B 0,C 180,E1 -14234.325,E2 -14234.325} C_VEL
LIN {X 0,Y 340.839,Z 429.026,A -85,B 0,C 180,E1 -14238.467,E2 -14238.467} C_VEL
LIN {X 0,Y 340.755,Z 429.039,A -85,B 0,C 180,E1 -14241.857,E2 -14241.857} C_VEL
LIN {X 0,Y 340.774,Z 429.036,A -85,B 0,C 180,E1 -14245.665,E2 -14245.665} C_VEL
LIN {X 0,Y 340.729,Z 429.041,A -85,B 0,C 180,E1 -14248.321,E2 -14248.321} C_VEL
LIN {X 0,Y 340.699,Z 429.042,A -85,B 0,C 180,E1 -14251.045,E2 -14251.045} C_VEL
LIN {X 0,Y 340.72,Z 429.04,A -85,B 0,C 180,E1 -14255.279,E2 -14255.279} C_VEL
LIN {X 0,Y 340.712,Z 429.042,A -85,B 0,C 180,E1 -14258.387,E2 -14258.387} C_VEL
LIN {X 0,Y 340.701,Z 429.046,A -85,B 0,C 180,E1 -14262.046,E2 -14262.046} C_VEL
LIN {X 0,Y 340.655,Z 429.05,A -85,B 0,C 180,E1 -14266.227,E2 -14266.227} C_VEL
LIN {X 0,Y 340.691,Z 429.049,A -85,B 0,C 180,E1 -14269.753,E2 -14269.753} C_VEL
LIN {X 0,Y 340.708,Z 429.043,A -85,B 0,C 180,E1 -14273.259,E2 -14273.259} C_VEL
LIN {X 0,Y 340.697,Z 429.045,A -85,B 0,C 180,E1 -14276.154,E2 -14276.154} C_VEL
LIN {X 0,Y 340.778,Z 429.033,A -85,B 0,C 180,E1 -14280.333,E2 -14280.333} C_VEL
LIN {X 0,Y 340.808,Z 429.03,A -85,B 0,C 180,E1 -14283.021,E2 -14283.021} C_VEL
LIN {X 0,Y 340.732,Z 429.039,A -85,B 0,C 180,E1 -14286.928,E2 -14286.928} C_VEL
LIN {X 0,Y 340.798,Z 429.031,A -85,B 0,C 180,E1 -14290.734,E2 -14290.734} C_VEL
LIN {X 0,Y 340.843,Z 429.229,A -85,B 0,C 180,E1 -14293.125,E2 -14293.125} C_VEL
LIN {X 0,Y 344.384,Z 439.862,A -85,B 0,C 180,E1 -14294.106,E2 -14294.106} C_VEL
LIN {X 0,Y 347.536,Z 451.33,A -85,B 0,C 180,E1 -14295.358,E2 -14295.358} C_VEL
LIN {X 0,Y 346.711,Z 461.741,A -85,B 0,C 180,E1 -14296.521,E2 -14296.521} C_VEL
LIN {X 0,Y 345.626,Z 471.902,A -85,B 0,C 180,E1 -14297.922,E2 -14297.922} C_VEL
LIN {X 0,Y 344.545,Z 480.725,A -85,B 0,C 180,E1 -14299.422,E2 -14299.422} C_VEL
LIN {X 0,Y 343.57,Z 488.965,A -85,B 0,C 180,E1 -14301.175,E2 -14301.175} C_VEL
LIN {X 0,Y 342.642,Z 495.597,A -85,B 0,C 180,E1 -14302.931,E2 -14302.931} C_VEL
LIN {X 0,Y 342.176,Z 500.851,A -85,B 0,C 180,E1 -14304.697,E2 -14304.697} C_VEL
LIN {X 0,Y 341.557,Z 505.006,A -85,B 0,C 180,E1 -14306.461,E2 -14306.461} C_VEL
LIN {X 0,Y 341.244,Z 507.21,A -85,B 0,C 180,E1 -14307.64,E2 -14307.64} C_VEL
LIN {X 0,Y 341.035,Z 508.964,A -85,B 0,C 180,E1 -14308.819,E2 -14308.819} C_VEL
LIN {X 0,Y 340.914,Z 511.21,A -85,B 0,C 180,E1 -14311.182,E2 -14311.182} C_VEL
LIN {X 0,Y 340.813,Z 511.79,A -85,B 0,C 180,E1 -14312.364,E2 -14312.364} C_VEL
LIN {X 0,Y 340.696,Z 511.98,A -85,B 0,C 180,E1 -14313.548,E2 -14313.548} C_VEL
LIN {X 0,Y 341.047,Z 511.124,A -85,B 0,C 180,E1 -14315.914,E2 -14315.914} C_VEL
LIN {X 0,Y 341.408,Z 510.122,A -85,B 0,C 180,E1 -14317.095,E2 -14317.095} C_VEL
LIN {X 0,Y 341.895,Z 507.091,A -85,B 0,C 180,E1 -14319.356,E2 -14319.356} C_VEL
LIN {X 0,Y 342.616,Z 503.332,A -85,B 0,C 180,E1 -14321.237,E2 -14321.237} C_VEL
LIN {X 0,Y 343.37,Z 498.671,A -85,B 0,C 180,E1 -14323.012,E2 -14323.012} C_VEL
LIN {X 0,Y 344.221,Z 492.769,A -85,B 0,C 180,E1 -14324.787,E2 -14324.787} C_VEL
LIN {X 0,Y 345.245,Z 485.398,A -85,B 0,C 180,E1 -14326.559,E2 -14326.559} C_VEL
LIN {X 0,Y 346.387,Z 477.809,A -85,B 0,C 180,E1 -14328.024,E2 -14328.024} C_VEL
LIN {X 0,Y 347.542,Z 467.48,A -85,B 0,C 180,E1 -14329.645,E2 -14329.645} C_VEL
LIN {X 0,Y 348.705,Z 456.9,A -85,B 0,C 180,E1 -14330.962,E2 -14330.962} C_VEL
LIN {X 0,Y 348.963,Z 454.151,A -85,B 0,C 180,E1 -14331.255,E2 -14331.255} C_VEL
LIN {X 0,Y 346.051,Z 444.212,A -85,B 0,C 180,E1 -14332.473,E2 -14332.473} C_VEL
LIN {X 0,Y 342.418,Z 433.86,A -85,B 0,C 180,E1 -14333.576,E2 -14333.576} C_VEL
LIN {X 0,Y 340.75,Z 429.039,A -85,B 0,C 180,E1 -14334.041,E2 -14334.041} C_VEL
LIN {X 0,Y 340.783,Z 429.033,A -85,B 0,C 180,E1 -14337.526,E2 -14337.526} C_VEL
LIN {X 0,Y 340.708,Z 429.042,A -85,B 0,C 180,E1 -14341.044,E2 -14341.044} C_VEL
LIN {X 0,Y 340.722,Z 429.04,A -85,B 0,C 180,E1 -14345.279,E2 -14345.279} C_VEL
LIN {X 0,Y 340.714,Z 429.045,A -85,B 0,C 180,E1 -14348.386,E2 -14348.386} C_VEL
LIN {X 0,Y 340.703,Z 429.048,A -85,B 0,C 180,E1 -14352.046,E2 -14352.046} C_VEL
LIN {X 0,Y 340.656,Z 429.052,A -85,B 0,C 180,E1 -14356.227,E2 -14356.227} C_VEL
LIN {X 0,Y 340.692,Z 429.047,A -85,B 0,C 180,E1 -14359.753,E2 -14359.753} C_VEL
LIN {X 0,Y 340.709,Z 429.042,A -85,B 0,C 180,E1 -14363.258,E2 -14363.258} C_VEL
LIN {X 0,Y 340.715,Z 429.04,A -85,B 0,C 180,E1 -14364.606,E2 -14364.606} C_VEL
LIN {X 0,Y 340.099,Z 429.122,A -85,B 0,C 180,E1 -14365.593,E2 -14365.593} C_VEL
LIN {X 0,Y 337.285,Z 429.48,A -85,B 0,C 180,E1 -14367.198,E2 -14367.198} C_VEL
LIN {X 0,Y 334.858,Z 429.782,A -85,B 0,C 180,E1 -14368.498,E2 -14368.498} C_VEL
LIN {X 0,Y 333.795,Z 429.908,A -85,B 0,C 180,E1 -14369.503,E2 -14369.503} C_VEL
LIN {X 0,Y 333.699,Z 429.917,A -85,B 0,C 180,E1 -14369.844,E2 -14369.844} C_VEL
LIN {X 0,Y 333.739,Z 429.915,A -85,B 0,C 180,E1 -14373.754,E2 -14373.754} C_VEL
LIN {X 0,Y 333.661,Z 429.925,A -85,B 0,C 180,E1 -14377.719,E2 -14377.719} C_VEL
LIN {X 0,Y 333.799,Z 429.907,A -85,B 0,C 180,E1 -14381.589,E2 -14381.589} C_VEL
LIN {X 0,Y 333.815,Z 430,A -85,B 0,C 180,E1 -14382.778,E2 -14382.778} C_VEL
LIN {X 0,Y 336.871,Z 442.253,A -85,B 0,C 180,E1 -14383.896,E2 -14383.896} C_VEL
LIN {X 0,Y 337.909,Z 447.723,A -85,B 0,C 180,E1 -14384.467,E2 -14384.467} C_VEL
LIN {X 0,Y 337.07,Z 459.838,A -85,B 0,C 180,E1 -14385.818,E2 -14385.818} C_VEL
LIN {X 0,Y 336.419,Z 470.686,A -85,B 0,C 180,E1 -14387.329,E2 -14387.329} C_VEL
LIN {X 0,Y 335.65,Z 479.647,A -85,B 0,C 180,E1 -14388.832,E2 -14388.832} C_VEL
LIN {X 0,Y 335.033,Z 488.63,A -85,B 0,C 180,E1 -14390.672,E2 -14390.672} C_VEL
LIN {X 0,Y 334.417,Z 496.746,A -85,B 0,C 180,E1 -14392.756,E2 -14392.756} C_VEL
LIN {X 0,Y 334.082,Z 502.349,A -85,B 0,C 180,E1 -14394.568,E2 -14394.568} C_VEL
LIN {X 0,Y 333.582,Z 506.802,A -85,B 0,C 180,E1 -14396.376,E2 -14396.376} C_VEL
LIN {X 0,Y 333.788,Z 509.108,A -85,B 0,C 180,E1 -14397.586,E2 -14397.586} C_VEL
LIN {X 0,Y 333.715,Z 511.043,A -85,B 0,C 180,E1 -14398.793,E2 -14398.793} C_VEL
LIN {X 0,Y 333.867,Z 512.538,A -85,B 0,C 180,E1 -14400,E2 -14400} C_VEL
LIN {X 0,Y 334.113,Z 514.267,A -85,B 0,C 180,E1 -14402.411,E2 -14402.411} C_VEL
LIN {X 0,Y 334.329,Z 514.545,A -85,B 0,C 180,E1 -14403.616,E2 -14403.616} C_VEL
LIN {X 0,Y 334.964,Z 513.824,A -85,B 0,C 180,E1 -14406.022,E2 -14406.022} C_VEL
LIN {X 0,Y 335.391,Z 512.892,A -85,B 0,C 180,E1 -14407.223,E2 -14407.223} C_VEL
LIN {X 0,Y 335.979,Z 511.497,A -85,B 0,C 180,E1 -14408.42,E2 -14408.42} C_VEL
LIN {X 0,Y 336.935,Z 508.615,A -85,B 0,C 180,E1 -14410.212,E2 -14410.212} C_VEL
LIN {X 0,Y 338.118,Z 504.663,A -85,B 0,C 180,E1 -14411.997,E2 -14411.997} C_VEL
LIN {X 0,Y 339.429,Z 499.631,A -85,B 0,C 180,E1 -14413.775,E2 -14413.775} C_VEL
LIN {X 0,Y 340.925,Z 493.334,A -85,B 0,C 180,E1 -14415.544,E2 -14415.544} C_VEL
LIN {X 0,Y 342.692,Z 485.454,A -85,B 0,C 180,E1 -14417.3,E2 -14417.3} C_VEL
LIN {X 0,Y 344.626,Z 475.748,A -85,B 0,C 180,E1 -14419.044,E2 -14419.044} C_VEL
LIN {X 0,Y 346.402,Z 466.087,A -85,B 0,C 180,E1 -14420.43,E2 -14420.43} C_VEL
LIN {X 0,Y 347.111,Z 461.895,A -85,B 0,C 180,E1 -14420.949,E2 -14420.949} C_VEL
LIN {X 0,Y 344.677,Z 453.151,A -85,B 0,C 180,E1 -14422.449,E2 -14422.449} C_VEL
LIN {X 0,Y 340.041,Z 442,A -85,B 0,C 180,E1 -14424.416,E2 -14424.416} C_VEL
LIN {X 0,Y 335.872,Z 434.176,A -85,B 0,C 180,E1 -14425.873,E2 -14425.873} C_VEL
LIN {X 0,Y 334.931,Z 433.072,A -85,B 0,C 180,E1 -14426.145,E2 -14426.145} C_VEL
LIN {X 0,Y 333.802,Z 430.235,A -85,B 0,C 180,E1 -14426.598,E2 -14426.598} C_VEL
LIN {X 0,Y 333.752,Z 429.912,A -85,B 0,C 180,E1 -14426.666,E2 -14426.666} C_VEL
LIN {X 0,Y 333.7,Z 429.918,A -85,B 0,C 180,E1 -14430.362,E2 -14430.362} C_VEL
LIN {X 0,Y 333.688,Z 429.92,A -85,B 0,C 180,E1 -14434.774,E2 -14434.774} C_VEL
LIN {X 0,Y 333.655,Z 429.921,A -85,B 0,C 180,E1 -14437.651,E2 -14437.651} C_VEL
LIN {X 0,Y 333.725,Z 430.103,A -85,B 0,C 180,E1 -14441.962,E2 -14441.962} C_VEL
LIN {X 0,Y 335.263,Z 437.587,A -85,B 0,C 180,E1 -14445.457,E2 -14445.457} C_VEL
LIN {X 0,Y 336.755,Z 444.939,A -85,B 0,C 180,E1 -14448.704,E2 -14448.704} C_VEL
LIN {X 0,Y 337.936,Z 451.436,A -85,B 0,C 180,E1 -14451.398,E2 -14451.398} C_VEL
LIN {X 0,Y 338.118,Z 453.391,A -85,B 0,C 180,E1 -14452.172,E2 -14452.172} C_VEL
LIN {X 0,Y 336.768,Z 462.986,A -85,B 0,C 180,E1 -14455.704,E2 -14455.704} C_VEL
LIN {X 0,Y 335.578,Z 472.616,A -85,B 0,C 180,E1 -14459.167,E2 -14459.167} C_VEL
LIN {X 0,Y 334.636,Z 481.968,A -85,B 0,C 180,E1 -14462.481,E2 -14462.481} C_VEL
LIN {X 0,Y 334.073,Z 488.058,A -85,B 0,C 180,E1 -14464.628,E2 -14464.628} C_VEL
LIN {X 0,Y 334.924,Z 492.758,A -85,B 0,C 180,E1 -14465.055,E2 -14465.055} C_VEL
LIN {X 0,Y 337.068,Z 503.628,A -85,B 0,C 180,E1 -14466.1,E2 -14466.1} C_VEL
LIN {X 0,Y 338.871,Z 518.463,A -85,B 0,C 180,E1 -14467.556,E2 -14467.556} C_VEL
LIN {X 0,Y 339.097,Z 528.357,A -85,B 0,C 180,E1 -14468.556,E2 -14468.556} C_VEL
LIN {X 0,Y 338.543,Z 542.443,A -85,B 0,C 180,E1 -14470.127,E2 -14470.127} C_VEL
LIN {X 0,Y 337.526,Z 556.093,A -85,B 0,C 180,E1 -14471.957,E2 -14471.957} C_VEL
LIN {X 0,Y 335.135,Z 571.606,A -85,B 0,C 180,E1 -14474.395,E2 -14474.395} C_VEL
LIN {X 0,Y 334.152,Z 580.063,A -85,B 0,C 180,E1 -14476.003,E2 -14476.003} C_VEL
LIN {X 0,Y 333.273,Z 587.837,A -85,B 0,C 180,E1 -14477.826,E2 -14477.826} C_VEL
LIN {X 0,Y 332.743,Z 594.145,A -85,B 0,C 180,E1 -14479.657,E2 -14479.657} C_VEL
LIN {X 0,Y 332.649,Z 599.212,A -85,B 0,C 180,E1 -14481.495,E2 -14481.495} C_VEL
LIN {X 0,Y 332.716,Z 602.75,A -85,B 0,C 180,E1 -14483.116,E2 -14483.116} C_VEL
LIN {X 0,Y 332.956,Z 606.044,A -85,B 0,C 180,E1 -14485.156,E2 -14485.156} C_VEL
LIN {X 0,Y 333.092,Z 607.425,A -85,B 0,C 180,E1 -14486.371,E2 -14486.371} C_VEL
LIN {X 0,Y 333.172,Z 608.387,A -85,B 0,C 180,E1 -14487.582,E2 -14487.582} C_VEL
LIN {X 0,Y 333.539,Z 608.945,A -85,B 0,C 180,E1 -14488.792,E2 -14488.792} C_VEL
LIN {X 0,Y 333.623,Z 609.039,A -85,B 0,C 180,E1 -14490,E2 -14490} C_VEL
LIN {X 0,Y 333.554,Z 608.708,A -85,B 0,C 180,E1 -14491.207,E2 -14491.207} C_VEL
LIN {X 0,Y 333.222,Z 607.933,A -85,B 0,C 180,E1 -14492.417,E2 -14492.417} C_VEL
LIN {X 0,Y 333.14,Z 606.749,A -85,B 0,C 180,E1 -14493.628,E2 -14493.628} C_VEL
LIN {X 0,Y 332.946,Z 604.144,A -85,B 0,C 180,E1 -14495.45,E2 -14495.45} C_VEL
LIN {X 0,Y 332.738,Z 600.476,A -85,B 0,C 180,E1 -14497.28,E2 -14497.28} C_VEL
LIN {X 0,Y 332.727,Z 595.686,A -85,B 0,C 180,E1 -14499.115,E2 -14499.115} C_VEL
LIN {X 0,Y 332.93,Z 589.629,A -85,B 0,C 180,E1 -14500.952,E2 -14500.952} C_VEL
LIN {X 0,Y 333.506,Z 582.118,A -85,B 0,C 180,E1 -14502.783,E2 -14502.783} C_VEL
LIN {X 0,Y 334.012,Z 576.175,A -85,B 0,C 180,E1 -14504.002,E2 -14504.002} C_VEL
LIN {X 0,Y 335.072,Z 567.342,A -85,B 0,C 180,E1 -14505.511,E2 -14505.511} C_VEL
LIN {X 0,Y 336.215,Z 556.475,A -85,B 0,C 180,E1 -14507.016,E2 -14507.016} C_VEL
LIN {X 0,Y 336.685,Z 551.364,A -85,B 0,C 180,E1 -14507.618,E2 -14507.618} C_VEL
LIN {X 0,Y 336.593,Z 540.718,A -85,B 0,C 180,E1 -14508.725,E2 -14508.725} C_VEL
LIN {X 0,Y 336.299,Z 528.939,A -85,B 0,C 180,E1 -14509.708,E2 -14509.708} C_VEL
LIN {X 0,Y 335.403,Z 515.288,A -85,B 0,C 180,E1 -14510.587,E2 -14510.587} C_VEL
LIN {X 0,Y 333.821,Z 501.669,A -85,B 0,C 180,E1 -14511.236,E2 -14511.236} C_VEL
LIN {X 0,Y 333.21,Z 497.03,A -85,B 0,C 180,E1 -14511.426,E2 -14511.426} C_VEL
LIN {X 0,Y 333.978,Z 484.905,A -85,B 0,C 180,E1 -14515.623,E2 -14515.623} C_VEL
LIN {X 0,Y 334.953,Z 473.66,A -85,B 0,C 180,E1 -14519.543,E2 -14519.543} C_VEL
LIN {X 0,Y 336.084,Z 463.152,A -85,B 0,C 180,E1 -14523.232,E2 -14523.232} C_VEL
LIN {X 0,Y 337.408,Z 452.224,A -85,B 0,C 180,E1 -14527.16,E2 -14527.16} C_VEL
LIN {X 0,Y 337.47,Z 449.661,A -85,B 0,C 180,E1 -14528.12,E2 -14528.12} C_VEL
LIN {X 0,Y 336.115,Z 442.059,A -85,B 0,C 180,E1 -14531.172,E2 -14531.172} C_VEL
LIN {X 0,Y 334.595,Z 434.399,A -85,B 0,C 180,E1 -14534.426,E2 -14534.426} C_VEL
LIN {X 0,Y 333.648,Z 429.931,A -85,B 0,C 180,E1 -14536.48,E2 -14536.48} C_VEL
LIN {X 0,Y 333.648,Z 429.923,A -85,B 0,C 180,E1 -14539.315,E2 -14539.315} C_VEL
LIN {X 0,Y 333.667,Z 429.919,A -85,B 0,C 180,E1 -14543.167,E2 -14543.167} C_VEL
LIN {X 0,Y 333.639,Z 429.924,A -85,B 0,C 180,E1 -14546.792,E2 -14546.792} C_VEL
LIN {X 0,Y 333.694,Z 429.918,A -85,B 0,C 180,E1 -14549.713,E2 -14549.713} C_VEL
LIN {X 0,Y 333.74,Z 429.913,A -85,B 0,C 180,E1 -14552.401,E2 -14552.401} C_VEL
LIN {X 0,Y 333.727,Z 429.911,A -85,B 0,C 180,E1 -14555.091,E2 -14555.091} C_VEL
LIN {X 0,Y 333.687,Z 429.917,A -85,B 0,C 180,E1 -14559.02,E2 -14559.02} C_VEL
LIN {X 0,Y 333.795,Z 429.905,A -85,B 0,C 180,E1 -14561.59,E2 -14561.59} C_VEL
LIN {X 0,Y 333.809,Z 429.903,A -85,B 0,C 180,E1 -14565.577,E2 -14565.577} C_VEL
LIN {X 0,Y 333.838,Z 429.898,A -85,B 0,C 180,E1 -14569.078,E2 -14569.078} C_VEL
LIN {X 0,Y 333.996,Z 429.879,A -85,B 0,C 180,E1 -14572.747,E2 -14572.747} C_VEL
LIN {X 0,Y 333.812,Z 429.901,A -85,B 0,C 180,E1 -14575.169,E2 -14575.169} C_VEL
LIN {X 0,Y 334.109,Z 429.865,A -85,B 0,C 180,E1 -14577.589,E2 -14577.589} C_VEL
LIN {X 0,Y 334.268,Z 429.85,A -85,B 0,C 180,E1 -14580,E2 -14580} C_VEL
LIN {X 0,Y 334.106,Z 429.866,A -85,B 0,C 180,E1 -14582.411,E2 -14582.411} C_VEL
LIN {X 0,Y 334.027,Z 429.873,A -85,B 0,C 180,E1 -14587.253,E2 -14587.253} C_VEL
LIN {X 0,Y 333.835,Z 429.897,A -85,B 0,C 180,E1 -14590.922,E2 -14590.922} C_VEL
LIN {X 0,Y 333.809,Z 429.901,A -85,B 0,C 180,E1 -14594.634,E2 -14594.634} C_VEL
LIN {X 0,Y 333.798,Z 429.902,A -85,B 0,C 180,E1 -14598.656,E2 -14598.656} C_VEL
LIN {X 0,Y 333.693,Z 429.914,A -85,B 0,C 180,E1 -14602.278,E2 -14602.278} C_VEL
LIN {X 0,Y 333.736,Z 429.913,A -85,B 0,C 180,E1 -14606.247,E2 -14606.247} C_VEL
LIN {X 0,Y 333.691,Z 429.916,A -85,B 0,C 180,E1 -14608.974,E2 -14608.974} C_VEL
LIN {X 0,Y 333.647,Z 429.918,A -85,B 0,C 180,E1 -14612.588,E2 -14612.588} C_VEL
LIN {X 0,Y 333.678,Z 429.92,A -85,B 0,C 180,E1 -14616.139,E2 -14616.139} C_VEL
LIN {X 0,Y 333.649,Z 429.922,A -85,B 0,C 180,E1 -14619.193,E2 -14619.193} C_VEL
LIN {X 0,Y 333.634,Z 429.923,A -85,B 0,C 180,E1 -14622.5,E2 -14622.5} C_VEL
LIN {X 0,Y 333.6,Z 429.931,A -85,B 0,C 180,E1 -14625.956,E2 -14625.956} C_VEL
LIN {X 0,Y 333.649,Z 429.922,A -85,B 0,C 180,E1 -14629.316,E2 -14629.316} C_VEL
LIN {X 0,Y 333.668,Z 429.919,A -85,B 0,C 180,E1 -14633.168,E2 -14633.168} C_VEL
LIN {X 0,Y 333.644,Z 429.921,A -85,B 0,C 180,E1 -14636.793,E2 -14636.793} C_VEL
LIN {X 0,Y 333.707,Z 429.919,A -85,B 0,C 180,E1 -14639.71,E2 -14639.71} C_VEL
LIN {X 0,Y 333.747,Z 429.909,A -85,B 0,C 180,E1 -14642.402,E2 -14642.402} C_VEL
LIN {X 0,Y 333.73,Z 429.911,A -85,B 0,C 180,E1 -14645.091,E2 -14645.091} C_VEL
LIN {X 0,Y 333.69,Z 429.917,A -85,B 0,C 180,E1 -14649.02,E2 -14649.02} C_VEL
LIN {X 0,Y 333.794,Z 429.904,A -85,B 0,C 180,E1 -14652.62,E2 -14652.62} C_VEL
LIN {X 0,Y 333.791,Z 430.015,A -85,B 0,C 180,E1 -14652.698,E2 -14652.698} C_VEL
LIN {X 0,Y 337.594,Z 441.481,A -85,B 0,C 180,E1 -14653.786,E2 -14653.786} C_VEL
LIN {X 0,Y 340.725,Z 452.699,A -85,B 0,C 180,E1 -14655.059,E2 -14655.059} C_VEL
LIN {X 0,Y 339.794,Z 464.228,A -85,B 0,C 180,E1 -14656.399,E2 -14656.399} C_VEL
LIN {X 0,Y 338.672,Z 474.185,A -85,B 0,C 180,E1 -14657.835,E2 -14657.835} C_VEL
LIN {X 0,Y 337.667,Z 481.931,A -85,B 0,C 180,E1 -14659.204,E2 -14659.204} C_VEL
LIN {X 0,Y 336.646,Z 490.125,A -85,B 0,C 180,E1 -14660.992,E2 -14660.992} C_VEL
LIN {X 0,Y 335.689,Z 496.729,A -85,B 0,C 180,E1 -14662.784,E2 -14662.784} C_VEL
LIN {X 0,Y 335.203,Z 501.958,A -85,B 0,C 180,E1 -14664.586,E2 -14664.586} C_VEL
LIN {X 0,Y 334.552,Z 506.093,A -85,B 0,C 180,E1 -14666.387,E2 -14666.387} C_VEL
LIN {X 0,Y 334.228,Z 508.286,A -85,B 0,C 180,E1 -14667.59,E2 -14667.59} C_VEL
LIN {X 0,Y 334.013,Z 510.02,A -85,B 0,C 180,E1 -14668.795,E2 -14668.795} C_VEL
LIN {X 0,Y 333.894,Z 512.245,A -85,B 0,C 180,E1 -14671.206,E2 -14671.206} C_VEL
LIN {X 0,Y 333.789,Z 512.816,A -85,B 0,C 180,E1 -14672.414,E2 -14672.414} C_VEL
LIN {X 0,Y 333.673,Z 512.987,A -85,B 0,C 180,E1 -14673.623,E2 -14673.623} C_VEL
LIN {X 0,Y 334.052,Z 512.112,A -85,B 0,C 180,E1 -14676.039,E2 -14676.039} C_VEL
LIN {X 0,Y 334.428,Z 511.1,A -85,B 0,C 180,E1 -14677.244,E2 -14677.244} C_VEL
LIN {X 0,Y 334.961,Z 508.04,A -85,B 0,C 180,E1 -14679.55,E2 -14679.55} C_VEL
LIN {X 0,Y 335.72,Z 504.256,A -85,B 0,C 180,E1 -14681.471,E2 -14681.471} C_VEL
LIN {X 0,Y 336.49,Z 499.576,A -85,B 0,C 180,E1 -14683.283,E2 -14683.283} C_VEL
LIN {X 0,Y 337.403,Z 493.647,A -85,B 0,C 180,E1 -14685.092,E2 -14685.092} C_VEL
LIN {X 0,Y 338.5,Z 486.243,A -85,B 0,C 180,E1 -14686.898,E2 -14686.898} C_VEL
LIN {X 0,Y 339.699,Z 478.613,A -85,B 0,C 180,E1 -14688.392,E2 -14688.392} C_VEL
LIN {X 0,Y 340.908,Z 468.23,A -85,B 0,C 180,E1 -14690.044,E2 -14690.044} C_VEL
LIN {X 0,Y 342.061,Z 458.069,A -85,B 0,C 180,E1 -14691.331,E2 -14691.331} C_VEL
LIN {X 0,Y 342.237,Z 456.37,A -85,B 0,C 180,E1 -14691.519,E2 -14691.519} C_VEL
LIN {X 0,Y 340.046,Z 448.136,A -85,B 0,C 180,E1 -14692.577,E2 -14692.577} C_VEL
LIN {X 0,Y 336.307,Z 437.122,A -85,B 0,C 180,E1 -14693.824,E2 -14693.824} C_VEL
LIN {X 0,Y 333.722,Z 429.914,A -85,B 0,C 180,E1 -14694.541,E2 -14694.541} C_VEL
LIN {X 0,Y 333.725,Z 429.913,A -85,B 0,C 180,E1 -14697.81,E2 -14697.81} C_VEL
LIN {X 0,Y 333.701,Z 429.92,A -85,B 0,C 180,E1 -14700.362,E2 -14700.362} C_VEL
LIN {X 0,Y 333.678,Z 429.919,A -85,B 0,C 180,E1 -14704.659,E2 -14704.659} C_VEL
LIN {X 0,Y 333.656,Z 429.922,A -85,B 0,C 180,E1 -14707.651,E2 -14707.651} C_VEL
LIN {X 0,Y 333.65,Z 429.922,A -85,B 0,C 180,E1 -14710.767,E2 -14710.767} C_VEL
LIN {X 0,Y 333.598,Z 429.932,A -85,B 0,C 180,E1 -14714.251,E2 -14714.251} C_VEL
LIN {X 0,Y 333.646,Z 429.923,A -85,B 0,C 180,E1 -14717.619,E2 -14717.619} C_VEL
LIN {X 0,Y 333.656,Z 429.92,A -85,B 0,C 180,E1 -14721.202,E2 -14721.202} C_VEL
LIN {X 0,Y 333.662,Z 429.919,A -85,B 0,C 180,E1 -14724.609,E2 -14724.609} C_VEL
LIN {X 0,Y 333.638,Z 429.925,A -85,B 0,C 180,E1 -14728.222,E2 -14728.222} C_VEL
LIN {X 0,Y 333.699,Z 429.917,A -85,B 0,C 180,E1 -14729.844,E2 -14729.844} C_VEL
LIN {X 0,Y 333.013,Z 430,A -85,B 0,C 180,E1 -14730.852,E2 -14730.852} C_VEL
LIN {X 0,Y 330.18,Z 430.354,A -85,B 0,C 180,E1 -14732.493,E2 -14732.493} C_VEL
LIN {X 0,Y 327.785,Z 430.657,A -85,B 0,C 180,E1 -14733.821,E2 -14733.821} C_VEL
LIN {X 0,Y 326.746,Z 430.781,A -85,B 0,C 180,E1 -14734.849,E2 -14734.849} C_VEL
LIN {X 0,Y 326.655,Z 430.792,A -85,B 0,C 180,E1 -14735.197,E2 -14735.197} C_VEL
LIN {X 0,Y 326.624,Z 430.796,A -85,B 0,C 180,E1 -14738.543,E2 -14738.543} C_VEL
LIN {X 0,Y 326.788,Z 430.776,A -85,B 0,C 180,E1 -14742.521,E2 -14742.521} C_VEL
LIN {X 0,Y 330.369,Z 445.402,A -85,B 0,C 180,E1 -14743.945,E2 -14743.945} C_VEL
LIN {X 0,Y 330.932,Z 448.611,A -85,B 0,C 180,E1 -14744.29,E2 -14744.29} C_VEL
LIN {X 0,Y 330.076,Z 460.739,A -85,B 0,C 180,E1 -14745.669,E2 -14745.669} C_VEL
LIN {X 0,Y 329.479,Z 470.615,A -85,B 0,C 180,E1 -14747.057,E2 -14747.057} C_VEL
LIN {X 0,Y 328.57,Z 481.365,A -85,B 0,C 180,E1 -14748.901,E2 -14748.901} C_VEL
LIN {X 0,Y 328.015,Z 489.283,A -85,B 0,C 180,E1 -14750.563,E2 -14750.563} C_VEL
LIN {X 0,Y 327.383,Z 497.148,A -85,B 0,C 180,E1 -14752.599,E2 -14752.599} C_VEL
LIN {X 0,Y 327.036,Z 502.904,A -85,B 0,C 180,E1 -14754.45,E2 -14754.45} C_VEL
LIN {X 0,Y 326.536,Z 507.504,A -85,B 0,C 180,E1 -14756.298,E2 -14756.298} C_VEL
LIN {X 0,Y 326.722,Z 510.98,A -85,B 0,C 180,E1 -14758.151,E2 -14758.151} C_VEL
LIN {X 0,Y 326.845,Z 513.484,A -85,B 0,C 180,E1 -14760,E2 -14760} C_VEL
LIN {X 0,Y 326.932,Z 514.628,A -85,B 0,C 180,E1 -14761.232,E2 -14761.232} C_VEL
LIN {X 0,Y 327.337,Z 515.71,A -85,B 0,C 180,E1 -14763.693,E2 -14763.693} C_VEL
LIN {X 0,Y 327.638,Z 515.656,A -85,B 0,C 180,E1 -14764.922,E2 -14764.922} C_VEL
LIN {X 0,Y 328.511,Z 514.282,A -85,B 0,C 180,E1 -14767.375,E2 -14767.375} C_VEL
LIN {X 0,Y 329.141,Z 512.989,A -85,B 0,C 180,E1 -14768.596,E2 -14768.596} C_VEL
LIN {X 0,Y 330.488,Z 509.11,A -85,B 0,C 180,E1 -14771.034,E2 -14771.034} C_VEL
LIN {X 0,Y 331.903,Z 504.804,A -85,B 0,C 180,E1 -14772.921,E2 -14772.921} C_VEL
LIN {X 0,Y 333.59,Z 498.686,A -85,B 0,C 180,E1 -14774.956,E2 -14774.956} C_VEL
LIN {X 0,Y 335.343,Z 491.866,A -85,B 0,C 180,E1 -14776.748,E2 -14776.748} C_VEL
LIN {X 0,Y 337.315,Z 483.455,A -85,B 0,C 180,E1 -14778.526,E2 -14778.526} C_VEL
LIN {X 0,Y 339.097,Z 474.842,A -85,B 0,C 180,E1 -14779.997,E2 -14779.997} C_VEL
LIN {X 0,Y 341.1,Z 464.584,A -85,B 0,C 180,E1 -14781.427,E2 -14781.427} C_VEL
LIN {X 0,Y 338.836,Z 456.23,A -85,B 0,C 180,E1 -14782.961,E2 -14782.961} C_VEL
LIN {X 0,Y 334.973,Z 446.449,A -85,B 0,C 180,E1 -14784.81,E2 -14784.81} C_VEL
LIN {X 0,Y 331.301,Z 439.206,A -85,B 0,C 180,E1 -14786.268,E2 -14786.268} C_VEL
LIN {X 0,Y 329.718,Z 436.463,A -85,B 0,C 180,E1 -14786.847,E2 -14786.847} C_VEL
LIN {X 0,Y 329.203,Z 435.331,A -85,B 0,C 180,E1 -14787.054,E2 -14787.054} C_VEL
LIN {X 0,Y 328.047,Z 434.114,A -85,B 0,C 180,E1 -14787.423,E2 -14787.423} C_VEL
LIN {X 0,Y 326.798,Z 431.473,A -85,B 0,C 180,E1 -14787.93,E2 -14787.93} C_VEL
LIN {X 0,Y 326.666,Z 430.792,A -85,B 0,C 180,E1 -14788.052,E2 -14788.052} C_VEL
LIN {X 0,Y 326.597,Z 430.802,A -85,B 0,C 180,E1 -14791.095,E2 -14791.095} C_VEL
LIN {X 0,Y 326.609,Z 430.8,A -85,B 0,C 180,E1 -14794.019,E2 -14794.019} C_VEL
LIN {X 0,Y 326.63,Z 430.796,A -85,B 0,C 180,E1 -14797.238,E2 -14797.238} C_VEL
LIN {X 0,Y 326.605,Z 430.796,A -85,B 0,C 180,E1 -14801.236,E2 -14801.236} C_VEL
LIN {X 0,Y 327.1,Z 433.039,A -85,B 0,C 180,E1 -14802.461,E2 -14802.461} C_VEL
LIN {X 0,Y 328.529,Z 440.092,A -85,B 0,C 180,E1 -14805.777,E2 -14805.777} C_VEL
LIN {X 0,Y 330.182,Z 448.196,A -85,B 0,C 180,E1 -14809.401,E2 -14809.401} C_VEL
LIN {X 0,Y 331.151,Z 454.464,A -85,B 0,C 180,E1 -14812.014,E2 -14812.014} C_VEL
LIN {X 0,Y 329.763,Z 464.009,A -85,B 0,C 180,E1 -14815.614,E2 -14815.614} C_VEL
LIN {X 0,Y 328.548,Z 473.491,A -85,B 0,C 180,E1 -14819.11,E2 -14819.11} C_VEL
LIN {X 0,Y 327.531,Z 482.888,A -85,B 0,C 180,E1 -14822.526,E2 -14822.526} C_VEL
LIN {X 0,Y 327.298,Z 485.532,A -85,B 0,C 180,E1 -14823.433,E2 -14823.433} C_VEL
LIN {X 0,Y 328.106,Z 489.92,A -85,B 0,C 180,E1 -14823.863,E2 -14823.863} C_VEL
LIN {X 0,Y 330.293,Z 500.5,A -85,B 0,C 180,E1 -14824.982,E2 -14824.982} C_VEL
LIN {X 0,Y 332.312,Z 516.007,A -85,B 0,C 180,E1 -14826.608,E2 -14826.608} C_VEL
LIN {X 0,Y 332.813,Z 527.097,A -85,B 0,C 180,E1 -14827.81,E2 -14827.81} C_VEL
LIN {X 0,Y 332.132,Z 540.87,A -85,B 0,C 180,E1 -14829.403,E2 -14829.403} C_VEL
LIN {X 0,Y 331.052,Z 554.45,A -85,B 0,C 180,E1 -14831.271,E2 -14831.271} C_VEL
LIN {X 0,Y 329.247,Z 564.779,A -85,B 0,C 180,E1 -14832.932,E2 -14832.932} C_VEL
LIN {X 0,Y 327.124,Z 579.14,A -85,B 0,C 180,E1 -14835.696,E2 -14835.696} C_VEL
LIN {X 0,Y 326.275,Z 586.904,A -85,B 0,C 180,E1 -14837.561,E2 -14837.561} C_VEL
LIN {X 0,Y 325.707,Z 593.194,A -85,B 0,C 180,E1 -14839.431,E2 -14839.431} C_VEL
LIN {X 0,Y 325.584,Z 598.245,A -85,B 0,C 180,E1 -14841.309,E2 -14841.309} C_VEL
LIN {X 0,Y 325.649,Z 602.009,A -85,B 0,C 180,E1 -14843.097,E2 -14843.097} C_VEL
LIN {X 0,Y 325.896,Z 605.054,A -85,B 0,C 180,E1 -14845.051,E2 -14845.051} C_VEL
LIN {X 0,Y 326.044,Z 606.431,A -85,B 0,C 180,E1 -14846.292,E2 -14846.292} C_VEL
LIN {X 0,Y 326.126,Z 607.387,A -85,B 0,C 180,E1 -14847.53,E2 -14847.53} C_VEL
LIN {X 0,Y 326.504,Z 607.935,A -85,B 0,C 180,E1 -14848.766,E2 -14848.766} C_VEL
LIN {X 0,Y 326.623,Z 608.027,A -85,B 0,C 180,E1 -14850,E2 -14850} C_VEL
LIN {X 0,Y 326.52,Z 607.684,A -85,B 0,C 180,E1 -14851.233,E2 -14851.233} C_VEL
LIN {X 0,Y 326.177,Z 606.9,A -85,B 0,C 180,E1 -14852.47,E2 -14852.47} C_VEL
LIN {X 0,Y 326.093,Z 605.7,A -85,B 0,C 180,E1 -14853.707,E2 -14853.707} C_VEL
LIN {X 0,Y 325.874,Z 603.076,A -85,B 0,C 180,E1 -14855.569,E2 -14855.569} C_VEL
